LIN {X 0,Y 368.899,Z 889.348,A -85,B 0,C 180,E1 -12566.461,E2 -12566.461} C_VEL
LIN {X 0,Y 368.899,Z 889.344,A -85,B 0,C 180,E1 -12569.043,E2 -12569.043} C_VEL
LIN {X 0,Y 368.91,Z 889.341,A -85,B 0,C 180,E1 -12571.557,E2 -12571.557} C_VEL
LIN {X 0,Y 368.887,Z 889.347,A -85,B 0,C 180,E1 -12575.219,E2 -12575.219} C_VEL
LIN {X 0,Y 368.898,Z 889.343,A -85,B 0,C 180,E1 -12577.602,E2 -12577.602} C_VEL
LIN {X 0,Y 368.909,Z 889.346,A -85,B 0,C 180,E1 -12581.103,E2 -12581.103} C_VEL
LIN {X 0,Y 368.931,Z 889.338,A -85,B 0,C 180,E1 -12584.532,E2 -12584.532} C_VEL
LIN {X 0,Y 369.059,Z 889.323,A -85,B 0,C 180,E1 -12586.79,E2 -12586.79} C_VEL
LIN {X 0,Y 369.059,Z 889.323,A -85,B 0,C 180,E1 -12590.131,E2 -12590.131} C_VEL
LIN {X 0,Y 369.157,Z 889.313,A -85,B 0,C 180,E1 -12593.44,E2 -12593.44} C_VEL
LIN {X 0,Y 369.292,Z 889.298,A -85,B 0,C 180,E1 -12597.818,E2 -12597.818} C_VEL
LIN {X 0,Y 369.204,Z 889.304,A -85,B 0,C 180,E1 -12601.09,E2 -12601.09} C_VEL
LIN {X 0,Y 369.292,Z 889.299,A -85,B 0,C 180,E1 -12602.181,E2 -12602.181} C_VEL
LIN {X 0,Y 369.157,Z 889.314,A -85,B 0,C 180,E1 -12606.559,E2 -12606.559} C_VEL
LIN {X 0,Y 369.058,Z 889.323,A -85,B 0,C 180,E1 -12609.868,E2 -12609.868} C_VEL
LIN {X 0,Y 369.04,Z 889.324,A -85,B 0,C 180,E1 -12613.772,E2 -12613.772} C_VEL
LIN {X 0,Y 368.955,Z 889.335,A -85,B 0,C 180,E1 -12617.744,E2 -12617.744} C_VEL
LIN {X 0,Y 368.91,Z 889.344,A -85,B 0,C 180,E1 -12621.22,E2 -12621.22} C_VEL
LIN {X 0,Y 368.906,Z 889.341,A -85,B 0,C 180,E1 -12623.872,E2 -12623.872} C_VEL
LIN {X 0,Y 368.856,Z 889.354,A -85,B 0,C 180,E1 -12627.212,E2 -12627.212} C_VEL
LIN {X 0,Y 368.892,Z 889.346,A -85,B 0,C 180,E1 -12629.692,E2 -12629.692} C_VEL
LIN {X 0,Y 368.895,Z 889.345,A -85,B 0,C 180,E1 -12633.042,E2 -12633.042} C_VEL
LIN {X 0,Y 368.91,Z 889.342,A -85,B 0,C 180,E1 -12636.197,E2 -12636.197} C_VEL
LIN {X 0,Y 368.872,Z 889.345,A -85,B 0,C 180,E1 -12638.957,E2 -12638.957} C_VEL
LIN {X 0,Y 368.858,Z 889.353,A -85,B 0,C 180,E1 -12642.005,E2 -12642.005} C_VEL
LIN {X 0,Y 368.872,Z 889.345,A -85,B 0,C 180,E1 -12645.174,E2 -12645.174} C_VEL
LIN {X 0,Y 368.86,Z 889.354,A -85,B 0,C 180,E1 -12648.174,E2 -12648.174} C_VEL
LIN {X 0,Y 368.873,Z 889.345,A -85,B 0,C 180,E1 -12651.366,E2 -12651.366} C_VEL
LIN {X 0,Y 368.931,Z 889.339,A -85,B 0,C 180,E1 -12655.145,E2 -12655.145} C_VEL
LIN {X 0,Y 368.895,Z 889.345,A -85,B 0,C 180,E1 -12659.043,E2 -12659.043} C_VEL
LIN {X 0,Y 368.883,Z 889.35,A -85,B 0,C 180,E1 -12662.79,E2 -12662.79} C_VEL
LIN {X 0,Y 368.943,Z 889.489,A -85,B 0,C 180,E1 -12663.316,E2 -12663.316} C_VEL
LIN {X 0,Y 371.115,Z 901.236,A -85,B 0,C 180,E1 -12666.566,E2 -12666.566} C_VEL
LIN {X 0,Y 370.607,Z 910.137,A -85,B 0,C 180,E1 -12668.881,E2 -12668.881} C_VEL
LIN {X 0,Y 369.569,Z 923.419,A -85,B 0,C 180,E1 -12672.286,E2 -12672.286} C_VEL
LIN {X 0,Y 369.237,Z 928.5,A -85,B 0,C 180,E1 -12673.547,E2 -12673.547} C_VEL
LIN {X 0,Y 372.227,Z 955.937,A -85,B 0,C 180,E1 -12674.334,E2 -12674.334} C_VEL
LIN {X 0,Y 371.384,Z 1006.743,A -85,B 0,C 180,E1 -12675.583,E2 -12675.583} C_VEL
LIN {X 0,Y 370.796,Z 1018.982,A -85,B 0,C 180,E1 -12676.085,E2 -12676.085} C_VEL
LIN {X 0,Y 370.446,Z 1028.911,A -85,B 0,C 180,E1 -12676.701,E2 -12676.701} C_VEL
LIN {X 0,Y 369.98,Z 1037.486,A -85,B 0,C 180,E1 -12677.382,E2 -12677.382} C_VEL
LIN {X 0,Y 369.472,Z 1045.773,A -85,B 0,C 180,E1 -12678.2,E2 -12678.2} C_VEL
LIN {X 0,Y 369.082,Z 1052.645,A -85,B 0,C 180,E1 -12679.023,E2 -12679.023} C_VEL
LIN {X 0,Y 368.68,Z 1058.484,A -85,B 0,C 180,E1 -12679.844,E2 -12679.844} C_VEL
LIN {X 0,Y 368.286,Z 1065.014,A -85,B 0,C 180,E1 -12680.942,E2 -12680.942} C_VEL
LIN {X 0,Y 367.983,Z 1070.432,A -85,B 0,C 180,E1 -12682.041,E2 -12682.041} C_VEL
LIN {X 0,Y 367.732,Z 1075.925,A -85,B 0,C 180,E1 -12683.415,E2 -12683.415} C_VEL
LIN {X 0,Y 367.595,Z 1081.012,A -85,B 0,C 180,E1 -12685.064,E2 -12685.064} C_VEL
LIN {X 0,Y 367.435,Z 1084.496,A -85,B 0,C 180,E1 -12686.71,E2 -12686.71} C_VEL
LIN {X 0,Y 367.453,Z 1086.131,A -85,B 0,C 180,E1 -12687.808,E2 -12687.808} C_VEL
LIN {X 0,Y 367.538,Z 1087.133,A -85,B 0,C 180,E1 -12688.904,E2 -12688.904} C_VEL
LIN {X 0,Y 367.52,Z 1087.577,A -85,B 0,C 180,E1 -12690,E2 -12690} C_VEL
LIN {X 0,Y 367.484,Z 1087.506,A -85,B 0,C 180,E1 -12691.096,E2 -12691.096} C_VEL
LIN {X 0,Y 367.412,Z 1086.92,A -85,B 0,C 180,E1 -12692.192,E2 -12692.192} C_VEL
LIN {X 0,Y 367.428,Z 1085.796,A -85,B 0,C 180,E1 -12693.289,E2 -12693.289} C_VEL
LIN {X 0,Y 367.571,Z 1082.946,A -85,B 0,C 180,E1 -12694.936,E2 -12694.936} C_VEL
LIN {X 0,Y 367.685,Z 1079.551,A -85,B 0,C 180,E1 -12696.315,E2 -12696.315} C_VEL
LIN {X 0,Y 367.978,Z 1075.132,A -85,B 0,C 180,E1 -12697.683,E2 -12697.683} C_VEL
LIN {X 0,Y 368.342,Z 1069.514,A -85,B 0,C 180,E1 -12699.056,E2 -12699.056} C_VEL
LIN {X 0,Y 368.948,Z 1062.566,A -85,B 0,C 180,E1 -12700.426,E2 -12700.426} C_VEL
LIN {X 0,Y 369.746,Z 1053.734,A -85,B 0,C 180,E1 -12701.79,E2 -12701.79} C_VEL
LIN {X 0,Y 370.374,Z 1046.059,A -85,B 0,C 180,E1 -12702.743,E2 -12702.743} C_VEL
LIN {X 0,Y 370.978,Z 1038.109,A -85,B 0,C 180,E1 -12703.558,E2 -12703.558} C_VEL
LIN {X 0,Y 371.559,Z 1030.04,A -85,B 0,C 180,E1 -12704.235,E2 -12704.235} C_VEL
LIN {X 0,Y 372.224,Z 1020.928,A -85,B 0,C 180,E1 -12704.837,E2 -12704.837} C_VEL
LIN {X 0,Y 372.916,Z 1010.324,A -85,B 0,C 180,E1 -12705.359,E2 -12705.359} C_VEL
LIN {X 0,Y 373.461,Z 995.486,A -85,B 0,C 180,E1 -12705.821,E2 -12705.821} C_VEL
LIN {X 0,Y 374.43,Z 954.567,A -85,B 0,C 180,E1 -12706.913,E2 -12706.913} C_VEL
LIN {X 0,Y 372.829,Z 940.302,A -85,B 0,C 180,E1 -12707.443,E2 -12707.443} C_VEL
LIN {X 0,Y 370.066,Z 925.912,A -85,B 0,C 180,E1 -12708.097,E2 -12708.097} C_VEL
LIN {X 0,Y 371.647,Z 911.366,A -85,B 0,C 180,E1 -12712.088,E2 -12712.088} C_VEL
LIN {X 0,Y 372.127,Z 906.885,A -85,B 0,C 180,E1 -12713.366,E2 -12713.366} C_VEL
LIN {X 0,Y 371.437,Z 901.089,A -85,B 0,C 180,E1 -12715.211,E2 -12715.211} C_VEL
LIN {X 0,Y 369.934,Z 893.844,A -85,B 0,C 180,E1 -12717.739,E2 -12717.739} C_VEL
LIN {X 0,Y 368.863,Z 889.353,A -85,B 0,C 180,E1 -12719.507,E2 -12719.507} C_VEL
LIN {X 0,Y 368.894,Z 889.349,A -85,B 0,C 180,E1 -12722.238,E2 -12722.238} C_VEL
LIN {X 0,Y 368.92,Z 889.346,A -85,B 0,C 180,E1 -12725,E2 -12725} C_VEL
LIN {X 0,Y 368.871,Z 889.35,A -85,B 0,C 180,E1 -12728.634,E2 -12728.634} C_VEL
LIN {X 0,Y 368.855,Z 889.351,A -85,B 0,C 180,E1 -12732.005,E2 -12732.005} C_VEL
LIN {X 0,Y 368.87,Z 889.349,A -85,B 0,C 180,E1 -12735.175,E2 -12735.175} C_VEL
LIN {X 0,Y 368.858,Z 889.352,A -85,B 0,C 180,E1 -12738.175,E2 -12738.175} C_VEL
LIN {X 0,Y 368.872,Z 889.349,A -85,B 0,C 180,E1 -12741.367,E2 -12741.367} C_VEL
LIN {X 0,Y 368.928,Z 889.341,A -85,B 0,C 180,E1 -12745.146,E2 -12745.146} C_VEL
LIN {X 0,Y 368.894,Z 889.347,A -85,B 0,C 180,E1 -12749.044,E2 -12749.044} C_VEL
LIN {X 0,Y 368.904,Z 889.345,A -85,B 0,C 180,E1 -12751.558,E2 -12751.558} C_VEL
LIN {X 0,Y 368.882,Z 889.354,A -85,B 0,C 180,E1 -12755.22,E2 -12755.22} C_VEL
LIN {X 0,Y 368.946,Z 889.49,A -85,B 0,C 180,E1 -12756.569,E2 -12756.569} C_VEL
LIN {X 0,Y 370.273,Z 896.019,A -85,B 0,C 180,E1 -12759.443,E2 -12759.443} C_VEL
LIN {X 0,Y 370.863,Z 900.746,A -85,B 0,C 180,E1 -12761.356,E2 -12761.356} C_VEL
LIN {X 0,Y 370.818,Z 902.644,A -85,B 0,C 180,E1 -12762.048,E2 -12762.048} C_VEL
LIN {X 0,Y 374.529,Z 916.761,A -85,B 0,C 180,E1 -12762.768,E2 -12762.768} C_VEL
LIN {X 0,Y 375.198,Z 921.412,A -85,B 0,C 180,E1 -12762.953,E2 -12762.953} C_VEL
LIN {X 0,Y 373.379,Z 979.291,A -85,B 0,C 180,E1 -12764.527,E2 -12764.527} C_VEL
LIN {X 0,Y 372.923,Z 991.072,A -85,B 0,C 180,E1 -12765.052,E2 -12765.052} C_VEL
LIN {X 0,Y 372.29,Z 1000.633,A -85,B 0,C 180,E1 -12765.655,E2 -12765.655} C_VEL
LIN {X 0,Y 371.8,Z 1008.981,A -85,B 0,C 180,E1 -12766.333,E2 -12766.333} C_VEL
LIN {X 0,Y 371.247,Z 1017.092,A -85,B 0,C 180,E1 -12767.148,E2 -12767.148} C_VEL
LIN {X 0,Y 370.556,Z 1024.861,A -85,B 0,C 180,E1 -12768.097,E2 -12768.097} C_VEL
LIN {X 0,Y 370.044,Z 1031.287,A -85,B 0,C 180,E1 -12769.052,E2 -12769.052} C_VEL
LIN {X 0,Y 369.282,Z 1038.862,A -85,B 0,C 180,E1 -12770.415,E2 -12770.415} C_VEL
LIN {X 0,Y 368.76,Z 1044.799,A -85,B 0,C 180,E1 -12771.783,E2 -12771.783} C_VEL
LIN {X 0,Y 368.34,Z 1050.206,A -85,B 0,C 180,E1 -12773.427,E2 -12773.427} C_VEL
LIN {X 0,Y 367.932,Z 1053.048,A -85,B 0,C 180,E1 -12774.52,E2 -12774.52} C_VEL
LIN {X 0,Y 367.798,Z 1055.276,A -85,B 0,C 180,E1 -12775.617,E2 -12775.617} C_VEL
LIN {X 0,Y 367.766,Z 1056.891,A -85,B 0,C 180,E1 -12776.714,E2 -12776.714} C_VEL
LIN {X 0,Y 367.665,Z 1057.898,A -85,B 0,C 180,E1 -12777.81,E2 -12777.81} C_VEL
LIN {X 0,Y 367.551,Z 1058.387,A -85,B 0,C 180,E1 -12778.905,E2 -12778.905} C_VEL
LIN {X 0,Y 367.504,Z 1058.367,A -85,B 0,C 180,E1 -12780.001,E2 -12780.001} C_VEL
LIN {X 0,Y 367.497,Z 1057.838,A -85,B 0,C 180,E1 -12781.096,E2 -12781.096} C_VEL
LIN {X 0,Y 367.517,Z 1056.751,A -85,B 0,C 180,E1 -12782.192,E2 -12782.192} C_VEL
LIN {X 0,Y 367.588,Z 1053.997,A -85,B 0,C 180,E1 -12783.837,E2 -12783.837} C_VEL
LIN {X 0,Y 367.744,Z 1051.48,A -85,B 0,C 180,E1 -12784.934,E2 -12784.934} C_VEL
LIN {X 0,Y 367.989,Z 1046.335,A -85,B 0,C 180,E1 -12786.581,E2 -12786.581} C_VEL
LIN {X 0,Y 368.218,Z 1042.025,A -85,B 0,C 180,E1 -12787.679,E2 -12787.679} C_VEL
LIN {X 0,Y 368.466,Z 1036.826,A -85,B 0,C 180,E1 -12788.778,E2 -12788.778} C_VEL
LIN {X 0,Y 368.906,Z 1030.558,A -85,B 0,C 180,E1 -12789.873,E2 -12789.873} C_VEL
LIN {X 0,Y 369.373,Z 1022.942,A -85,B 0,C 180,E1 -12790.969,E2 -12790.969} C_VEL
LIN {X 0,Y 369.855,Z 1014.814,A -85,B 0,C 180,E1 -12791.926,E2 -12791.926} C_VEL
LIN {X 0,Y 370.421,Z 1004.687,A -85,B 0,C 180,E1 -12792.882,E2 -12792.882} C_VEL
LIN {X 0,Y 370.87,Z 993.951,A -85,B 0,C 180,E1 -12793.633,E2 -12793.633} C_VEL
LIN {X 0,Y 371.104,Z 984.065,A -85,B 0,C 180,E1 -12794.148,E2 -12794.148} C_VEL
LIN {X 0,Y 371.472,Z 973.564,A -85,B 0,C 180,E1 -12794.518,E2 -12794.518} C_VEL
LIN {X 0,Y 372.416,Z 918.799,A -85,B 0,C 180,E1 -12795.838,E2 -12795.838} C_VEL
LIN {X 0,Y 369.303,Z 899.54,A -85,B 0,C 180,E1 -12796.448,E2 -12796.448} C_VEL
LIN {X 0,Y 369.477,Z 893.53,A -85,B 0,C 180,E1 -12798.363,E2 -12798.363} C_VEL
LIN {X 0,Y 369.004,Z 889.33,A -85,B 0,C 180,E1 -12799.76,E2 -12799.76} C_VEL
LIN {X 0,Y 368.906,Z 889.341,A -85,B 0,C 180,E1 -12803.873,E2 -12803.873} C_VEL
LIN {X 0,Y 368.857,Z 889.354,A -85,B 0,C 180,E1 -12807.213,E2 -12807.213} C_VEL
LIN {X 0,Y 368.893,Z 889.346,A -85,B 0,C 180,E1 -12809.693,E2 -12809.693} C_VEL
LIN {X 0,Y 368.897,Z 889.344,A -85,B 0,C 180,E1 -12813.043,E2 -12813.043} C_VEL
LIN {X 0,Y 368.913,Z 889.341,A -85,B 0,C 180,E1 -12816.198,E2 -12816.198} C_VEL
LIN {X 0,Y 368.874,Z 889.345,A -85,B 0,C 180,E1 -12818.958,E2 -12818.958} C_VEL
LIN {X 0,Y 368.86,Z 889.352,A -85,B 0,C 180,E1 -12822.006,E2 -12822.006} C_VEL
LIN {X 0,Y 368.874,Z 889.345,A -85,B 0,C 180,E1 -12825.175,E2 -12825.175} C_VEL
LIN {X 0,Y 368.863,Z 889.353,A -85,B 0,C 180,E1 -12828.175,E2 -12828.175} C_VEL
LIN {X 0,Y 368.877,Z 889.345,A -85,B 0,C 180,E1 -12831.367,E2 -12831.367} C_VEL
LIN {X 0,Y 368.934,Z 889.338,A -85,B 0,C 180,E1 -12835.146,E2 -12835.146} C_VEL
LIN {X 0,Y 368.899,Z 889.344,A -85,B 0,C 180,E1 -12839.044,E2 -12839.044} C_VEL
LIN {X 0,Y 368.91,Z 889.341,A -85,B 0,C 180,E1 -12841.558,E2 -12841.558} C_VEL
LIN {X 0,Y 368.925,Z 889.342,A -85,B 0,C 180,E1 -12845.222,E2 -12845.222} C_VEL
LIN {X 0,Y 368.924,Z 889.344,A -85,B 0,C 180,E1 -12848.981,E2 -12848.981} C_VEL
LIN {X 0,Y 368.957,Z 889.335,A -85,B 0,C 180,E1 -12852.256,E2 -12852.256} C_VEL
LIN {X 0,Y 369.017,Z 889.331,A -85,B 0,C 180,E1 -12855.665,E2 -12855.665} C_VEL
LIN {X 0,Y 369.013,Z 889.33,A -85,B 0,C 180,E1 -12859.021,E2 -12859.021} C_VEL
LIN {X 0,Y 369.12,Z 889.315,A -85,B 0,C 180,E1 -12862.341,E2 -12862.341} C_VEL
LIN {X 0,Y 369.117,Z 889.315,A -85,B 0,C 180,E1 -12864.537,E2 -12864.537} C_VEL
LIN {X 0,Y 369.295,Z 889.298,A -85,B 0,C 180,E1 -12867.819,E2 -12867.819} C_VEL
LIN {X 0,Y 369.206,Z 889.304,A -85,B 0,C 180,E1 -12871.091,E2 -12871.091} C_VEL
LIN {X 0,Y 369.294,Z 889.299,A -85,B 0,C 180,E1 -12872.182,E2 -12872.182} C_VEL
LIN {X 0,Y 369.159,Z 889.314,A -85,B 0,C 180,E1 -12876.559,E2 -12876.559} C_VEL
LIN {X 0,Y 369.061,Z 889.323,A -85,B 0,C 180,E1 -12879.869,E2 -12879.869} C_VEL
LIN {X 0,Y 369.043,Z 889.324,A -85,B 0,C 180,E1 -12883.772,E2 -12883.772} C_VEL
LIN {X 0,Y 368.958,Z 889.334,A -85,B 0,C 180,E1 -12887.745,E2 -12887.745} C_VEL
LIN {X 0,Y 368.913,Z 889.344,A -85,B 0,C 180,E1 -12891.221,E2 -12891.221} C_VEL
LIN {X 0,Y 368.909,Z 889.341,A -85,B 0,C 180,E1 -12893.872,E2 -12893.872} C_VEL
LIN {X 0,Y 368.86,Z 889.353,A -85,B 0,C 180,E1 -12897.212,E2 -12897.212} C_VEL
LIN {X 0,Y 368.896,Z 889.345,A -85,B 0,C 180,E1 -12899.692,E2 -12899.692} C_VEL
LIN {X 0,Y 368.9,Z 889.344,A -85,B 0,C 180,E1 -12903.042,E2 -12903.042} C_VEL
LIN {X 0,Y 368.89,Z 889.344,A -85,B 0,C 180,E1 -12904.117,E2 -12904.117} C_VEL
LIN {X 0,Y 368.239,Z 889.427,A -85,B 0,C 180,E1 -12905.029,E2 -12905.029} C_VEL
LIN {X 0,Y 365.381,Z 889.78,A -85,B 0,C 180,E1 -12906.512,E2 -12906.512} C_VEL
LIN {X 0,Y 362.952,Z 890.09,A -85,B 0,C 180,E1 -12907.711,E2 -12907.711} C_VEL
LIN {X 0,Y 361.911,Z 890.213,A -85,B 0,C 180,E1 -12908.639,E2 -12908.639} C_VEL
LIN {X 0,Y 361.829,Z 890.223,A -85,B 0,C 180,E1 -12908.953,E2 -12908.953} C_VEL
LIN {X 0,Y 361.833,Z 890.222,A -85,B 0,C 180,E1 -12912.83,E2 -12912.83} C_VEL
LIN {X 0,Y 361.817,Z 890.229,A -85,B 0,C 180,E1 -12915.947,E2 -12915.947} C_VEL
LIN {X 0,Y 361.813,Z 890.224,A -85,B 0,C 180,E1 -12919.249,E2 -12919.249} C_VEL
LIN {X 0,Y 361.864,Z 890.219,A -85,B 0,C 180,E1 -12922.981,E2 -12922.981} C_VEL
LIN {X 0,Y 361.861,Z 890.224,A -85,B 0,C 180,E1 -12926.631,E2 -12926.631} C_VEL
LIN {X 0,Y 361.85,Z 890.22,A -85,B 0,C 180,E1 -12929.669,E2 -12929.669} C_VEL
LIN {X 0,Y 361.857,Z 890.22,A -85,B 0,C 180,E1 -12933.467,E2 -12933.467} C_VEL
LIN {X 0,Y 361.863,Z 890.224,A -85,B 0,C 180,E1 -12937.142,E2 -12937.142} C_VEL
LIN {X 0,Y 361.849,Z 890.222,A -85,B 0,C 180,E1 -12940.72,E2 -12940.72} C_VEL
LIN {X 0,Y 361.89,Z 890.219,A -85,B 0,C 180,E1 -12943.063,E2 -12943.063} C_VEL
LIN {X 0,Y 362.002,Z 890.201,A -85,B 0,C 180,E1 -12946.527,E2 -12946.527} C_VEL
LIN {X 0,Y 361.996,Z 890.205,A -85,B 0,C 180,E1 -12949.936,E2 -12949.936} C_VEL
LIN {X 0,Y 362.121,Z 890.189,A -85,B 0,C 180,E1 -12953.312,E2 -12953.312} C_VEL
LIN {X 0,Y 362.254,Z 890.175,A -85,B 0,C 180,E1 -12957.776,E2 -12957.776} C_VEL
LIN {X 0,Y 362.175,Z 890.179,A -85,B 0,C 180,E1 -12961.111,E2 -12961.111} C_VEL
LIN {X 0,Y 362.254,Z 890.175,A -85,B 0,C 180,E1 -12962.223,E2 -12962.223} C_VEL
LIN {X 0,Y 362.121,Z 890.189,A -85,B 0,C 180,E1 -12966.687,E2 -12966.687} C_VEL
LIN {X 0,Y 361.995,Z 890.205,A -85,B 0,C 180,E1 -12970.063,E2 -12970.063} C_VEL
LIN {X 0,Y 361.982,Z 890.204,A -85,B 0,C 180,E1 -12973.886,E2 -12973.886} C_VEL
LIN {X 0,Y 361.886,Z 890.216,A -85,B 0,C 180,E1 -12978.103,E2 -12978.103} C_VEL
LIN {X 0,Y 361.853,Z 890.22,A -85,B 0,C 180,E1 -12981.655,E2 -12981.655} C_VEL
LIN {X 0,Y 361.859,Z 890.224,A -85,B 0,C 180,E1 -12985.295,E2 -12985.295} C_VEL
LIN {X 0,Y 361.856,Z 890.223,A -85,B 0,C 180,E1 -12989.073,E2 -12989.073} C_VEL
LIN {X 0,Y 361.847,Z 890.222,A -85,B 0,C 180,E1 -12992.944,E2 -12992.944} C_VEL
LIN {X 0,Y 361.863,Z 890.225,A -85,B 0,C 180,E1 -12995.637,E2 -12995.637} C_VEL
LIN {X 0,Y 361.824,Z 890.224,A -85,B 0,C 180,E1 -12999.017,E2 -12999.017} C_VEL
LIN {X 0,Y 361.828,Z 890.223,A -85,B 0,C 180,E1 -13002.83,E2 -13002.83} C_VEL
LIN {X 0,Y 361.813,Z 890.23,A -85,B 0,C 180,E1 -13005.947,E2 -13005.947} C_VEL
LIN {X 0,Y 361.809,Z 890.225,A -85,B 0,C 180,E1 -13009.249,E2 -13009.249} C_VEL
LIN {X 0,Y 361.86,Z 890.22,A -85,B 0,C 180,E1 -13012.981,E2 -13012.981} C_VEL
LIN {X 0,Y 361.856,Z 890.225,A -85,B 0,C 180,E1 -13016.631,E2 -13016.631} C_VEL
LIN {X 0,Y 361.845,Z 890.22,A -85,B 0,C 180,E1 -13019.669,E2 -13019.669} C_VEL
LIN {X 0,Y 361.879,Z 890.287,A -85,B 0,C 180,E1 -13023.145,E2 -13023.145} C_VEL
LIN {X 0,Y 364.001,Z 901.747,A -85,B 0,C 180,E1 -13026.382,E2 -13026.382} C_VEL
LIN {X 0,Y 363.896,Z 906.742,A -85,B 0,C 180,E1 -13027.718,E2 -13027.718} C_VEL
LIN {X 0,Y 362.776,Z 920.524,A -85,B 0,C 180,E1 -13031.332,E2 -13031.332} C_VEL
LIN {X 0,Y 362.246,Z 928.09,A -85,B 0,C 180,E1 -13033.3,E2 -13033.3} C_VEL
LIN {X 0,Y 365.281,Z 955.565,A -85,B 0,C 180,E1 -13034.116,E2 -13034.116} C_VEL
LIN {X 0,Y 364.371,Z 1006.424,A -85,B 0,C 180,E1 -13035.413,E2 -13035.413} C_VEL
LIN {X 0,Y 363.82,Z 1017.855,A -85,B 0,C 180,E1 -13035.884,E2 -13035.884} C_VEL
LIN {X 0,Y 363.4,Z 1028.918,A -85,B 0,C 180,E1 -13036.58,E2 -13036.58} C_VEL
LIN {X 0,Y 362.924,Z 1037.423,A -85,B 0,C 180,E1 -13037.274,E2 -13037.274} C_VEL
LIN {X 0,Y 362.418,Z 1045.665,A -85,B 0,C 180,E1 -13038.109,E2 -13038.109} C_VEL
LIN {X 0,Y 362.017,Z 1052.505,A -85,B 0,C 180,E1 -13038.947,E2 -13038.947} C_VEL
LIN {X 0,Y 361.548,Z 1059.189,A -85,B 0,C 180,E1 -13039.924,E2 -13039.924} C_VEL
LIN {X 0,Y 361.158,Z 1065.557,A -85,B 0,C 180,E1 -13041.044,E2 -13041.044} C_VEL
LIN {X 0,Y 360.886,Z 1070.836,A -85,B 0,C 180,E1 -13042.165,E2 -13042.165} C_VEL
LIN {X 0,Y 360.693,Z 1075.211,A -85,B 0,C 180,E1 -13043.286,E2 -13043.286} C_VEL
LIN {X 0,Y 360.51,Z 1080.389,A -85,B 0,C 180,E1 -13044.967,E2 -13044.967} C_VEL
LIN {X 0,Y 360.356,Z 1084.025,A -85,B 0,C 180,E1 -13046.646,E2 -13046.646} C_VEL
LIN {X 0,Y 360.359,Z 1085.689,A -85,B 0,C 180,E1 -13047.764,E2 -13047.764} C_VEL
LIN {X 0,Y 360.454,Z 1086.735,A -85,B 0,C 180,E1 -13048.883,E2 -13048.883} C_VEL
LIN {X 0,Y 360.456,Z 1087.245,A -85,B 0,C 180,E1 -13050,E2 -13050} C_VEL
LIN {X 0,Y 360.385,Z 1087.233,A -85,B 0,C 180,E1 -13051.117,E2 -13051.117} C_VEL
LIN {X 0,Y 360.314,Z 1086.702,A -85,B 0,C 180,E1 -13052.235,E2 -13052.235} C_VEL
LIN {X 0,Y 360.348,Z 1085.596,A -85,B 0,C 180,E1 -13053.354,E2 -13053.354} C_VEL
LIN {X 0,Y 360.488,Z 1082.825,A -85,B 0,C 180,E1 -13055.033,E2 -13055.033} C_VEL
LIN {X 0,Y 360.666,Z 1078.695,A -85,B 0,C 180,E1 -13056.714,E2 -13056.714} C_VEL
LIN {X 0,Y 360.999,Z 1074.143,A -85,B 0,C 180,E1 -13058.114,E2 -13058.114} C_VEL
LIN {X 0,Y 361.479,Z 1068.4,A -85,B 0,C 180,E1 -13059.512,E2 -13059.512} C_VEL
LIN {X 0,Y 362.14,Z 1061.248,A -85,B 0,C 180,E1 -13060.907,E2 -13060.907} C_VEL
LIN {X 0,Y 362.947,Z 1052.036,A -85,B 0,C 180,E1 -13062.298,E2 -13062.298} C_VEL
LIN {X 0,Y 363.677,Z 1044.075,A -85,B 0,C 180,E1 -13063.266,E2 -13063.266} C_VEL
LIN {X 0,Y 364.446,Z 1034.341,A -85,B 0,C 180,E1 -13064.233,E2 -13064.233} C_VEL
LIN {X 0,Y 365.322,Z 1023.496,A -85,B 0,C 180,E1 -13065.053,E2 -13065.053} C_VEL
LIN {X 0,Y 366.111,Z 1013.024,A -85,B 0,C 180,E1 -13065.623,E2 -13065.623} C_VEL
LIN {X 0,Y 366.578,Z 1003.239,A -85,B 0,C 180,E1 -13066.007,E2 -13066.007} C_VEL
LIN {X 0,Y 367.916,Z 955.498,A -85,B 0,C 180,E1 -13067.329,E2 -13067.329} C_VEL
LIN {X 0,Y 366.449,Z 941.662,A -85,B 0,C 180,E1 -13067.87,E2 -13067.87} C_VEL
LIN {X 0,Y 363.843,Z 928.167,A -85,B 0,C 180,E1 -13068.508,E2 -13068.508} C_VEL
LIN {X 0,Y 363.285,Z 925.477,A -85,B 0,C 180,E1 -13068.664,E2 -13068.664} C_VEL
LIN {X 0,Y 364.942,Z 911.374,A -85,B 0,C 180,E1 -13072.653,E2 -13072.653} C_VEL
LIN {X 0,Y 365.222,Z 907.458,A -85,B 0,C 180,E1 -13073.835,E2 -13073.835} C_VEL
LIN {X 0,Y 364.427,Z 901.823,A -85,B 0,C 180,E1 -13075.715,E2 -13075.715} C_VEL
LIN {X 0,Y 362.904,Z 894.732,A -85,B 0,C 180,E1 -13078.324,E2 -13078.324} C_VEL
LIN {X 0,Y 361.839,Z 890.227,A -85,B 0,C 180,E1 -13080.17,E2 -13080.17} C_VEL
LIN {X 0,Y 361.855,Z 890.227,A -85,B 0,C 180,E1 -13083.369,E2 -13083.369} C_VEL
LIN {X 0,Y 361.857,Z 890.224,A -85,B 0,C 180,E1 -13087.019,E2 -13087.019} C_VEL
LIN {X 0,Y 361.807,Z 890.227,A -85,B 0,C 180,E1 -13090.751,E2 -13090.751} C_VEL
LIN {X 0,Y 361.809,Z 890.231,A -85,B 0,C 180,E1 -13094.37,E2 -13094.37} C_VEL
LIN {X 0,Y 361.82,Z 890.227,A -85,B 0,C 180,E1 -13097.571,E2 -13097.571} C_VEL
LIN {X 0,Y 361.838,Z 890.226,A -85,B 0,C 180,E1 -13101.572,E2 -13101.572} C_VEL
LIN {X 0,Y 361.868,Z 890.222,A -85,B 0,C 180,E1 -13104.657,E2 -13104.657} C_VEL
LIN {X 0,Y 361.835,Z 890.227,A -85,B 0,C 180,E1 -13108.371,E2 -13108.371} C_VEL
LIN {X 0,Y 361.847,Z 890.226,A -85,B 0,C 180,E1 -13110.951,E2 -13110.951} C_VEL
LIN {X 0,Y 361.857,Z 890.227,A -85,B 0,C 180,E1 -13114.705,E2 -13114.705} C_VEL
LIN {X 0,Y 361.886,Z 890.418,A -85,B 0,C 180,E1 -13115.932,E2 -13115.932} C_VEL
LIN {X 0,Y 363.302,Z 897.119,A -85,B 0,C 180,E1 -13119.031,E2 -13119.031} C_VEL
LIN {X 0,Y 363.99,Z 902.06,A -85,B 0,C 180,E1 -13121.103,E2 -13121.103} C_VEL
LIN {X 0,Y 363.981,Z 903.044,A -85,B 0,C 180,E1 -13121.488,E2 -13121.488} C_VEL
LIN {X 0,Y 367.562,Z 915.604,A -85,B 0,C 180,E1 -13122.198,E2 -13122.198} C_VEL
LIN {X 0,Y 368.772,Z 921.813,A -85,B 0,C 180,E1 -13122.492,E2 -13122.492} C_VEL
LIN {X 0,Y 366.755,Z 980.697,A -85,B 0,C 180,E1 -13124.154,E2 -13124.154} C_VEL
LIN {X 0,Y 366.287,Z 992.208,A -85,B 0,C 180,E1 -13124.703,E2 -13124.703} C_VEL
LIN {X 0,Y 365.566,Z 1002.438,A -85,B 0,C 180,E1 -13125.385,E2 -13125.385} C_VEL
LIN {X 0,Y 364.916,Z 1011.91,A -85,B 0,C 180,E1 -13126.212,E2 -13126.212} C_VEL
LIN {X 0,Y 364.076,Z 1021.861,A -85,B 0,C 180,E1 -13127.316,E2 -13127.316} C_VEL
LIN {X 0,Y 363.31,Z 1030.516,A -85,B 0,C 180,E1 -13128.564,E2 -13128.564} C_VEL
LIN {X 0,Y 362.618,Z 1036.852,A -85,B 0,C 180,E1 -13129.673,E2 -13129.673} C_VEL
LIN {X 0,Y 362.121,Z 1042.099,A -85,B 0,C 180,E1 -13130.787,E2 -13130.787} C_VEL
LIN {X 0,Y 361.786,Z 1045.497,A -85,B 0,C 180,E1 -13131.623,E2 -13131.623} C_VEL
LIN {X 0,Y 361.42,Z 1049.962,A -85,B 0,C 180,E1 -13132.982,E2 -13132.982} C_VEL
LIN {X 0,Y 360.899,Z 1053.596,A -85,B 0,C 180,E1 -13134.413,E2 -13134.413} C_VEL
LIN {X 0,Y 360.73,Z 1055.75,A -85,B 0,C 180,E1 -13135.531,E2 -13135.531} C_VEL
LIN {X 0,Y 360.699,Z 1057.33,A -85,B 0,C 180,E1 -13136.649,E2 -13136.649} C_VEL
LIN {X 0,Y 360.591,Z 1058.296,A -85,B 0,C 180,E1 -13137.767,E2 -13137.767} C_VEL
LIN {X 0,Y 360.472,Z 1058.722,A -85,B 0,C 180,E1 -13138.883,E2 -13138.883} C_VEL
LIN {X 0,Y 360.423,Z 1058.638,A -85,B 0,C 180,E1 -13140.001,E2 -13140.001} C_VEL
LIN {X 0,Y 360.4,Z 1058.044,A -85,B 0,C 180,E1 -13141.118,E2 -13141.118} C_VEL
LIN {X 0,Y 360.42,Z 1056.916,A -85,B 0,C 180,E1 -13142.236,E2 -13142.236} C_VEL
LIN {X 0,Y 360.514,Z 1054.049,A -85,B 0,C 180,E1 -13143.913,E2 -13143.913} C_VEL
LIN {X 0,Y 360.715,Z 1049.844,A -85,B 0,C 180,E1 -13145.591,E2 -13145.591} C_VEL
LIN {X 0,Y 361.049,Z 1044.378,A -85,B 0,C 180,E1 -13147.213,E2 -13147.213} C_VEL
LIN {X 0,Y 361.337,Z 1037.934,A -85,B 0,C 180,E1 -13148.67,E2 -13148.67} C_VEL
LIN {X 0,Y 361.773,Z 1031.811,A -85,B 0,C 180,E1 -13149.787,E2 -13149.787} C_VEL
LIN {X 0,Y 362.24,Z 1024.366,A -85,B 0,C 180,E1 -13150.905,E2 -13150.905} C_VEL
LIN {X 0,Y 362.732,Z 1016.449,A -85,B 0,C 180,E1 -13151.88,E2 -13151.88} C_VEL
LIN {X 0,Y 363.163,Z 1008.15,A -85,B 0,C 180,E1 -13152.717,E2 -13152.717} C_VEL
LIN {X 0,Y 363.666,Z 997.731,A -85,B 0,C 180,E1 -13153.552,E2 -13153.552} C_VEL
LIN {X 0,Y 364.041,Z 986.186,A -85,B 0,C 180,E1 -13154.214,E2 -13154.214} C_VEL
LIN {X 0,Y 364.4,Z 975.683,A -85,B 0,C 180,E1 -13154.622,E2 -13154.622} C_VEL
LIN {X 0,Y 365.486,Z 919.722,A -85,B 0,C 180,E1 -13156.033,E2 -13156.033} C_VEL
LIN {X 0,Y 362.287,Z 899.844,A -85,B 0,C 180,E1 -13156.663,E2 -13156.663} C_VEL
LIN {X 0,Y 362.414,Z 893.862,A -85,B 0,C 180,E1 -13158.603,E2 -13158.603} C_VEL
LIN {X 0,Y 361.979,Z 890.205,A -85,B 0,C 180,E1 -13159.864,E2 -13159.864} C_VEL
LIN {X 0,Y 361.862,Z 890.218,A -85,B 0,C 180,E1 -13164.102,E2 -13164.102} C_VEL
LIN {X 0,Y 361.835,Z 890.223,A -85,B 0,C 180,E1 -13167.786,E2 -13167.786} C_VEL
LIN {X 0,Y 361.849,Z 890.225,A -85,B 0,C 180,E1 -13171.286,E2 -13171.286} C_VEL
LIN {X 0,Y 361.853,Z 890.22,A -85,B 0,C 180,E1 -13174.281,E2 -13174.281} C_VEL
LIN {X 0,Y 361.859,Z 890.221,A -85,B 0,C 180,E1 -13177.222,E2 -13177.222} C_VEL
LIN {X 0,Y 361.812,Z 890.225,A -85,B 0,C 180,E1 -13180.751,E2 -13180.751} C_VEL
LIN {X 0,Y 361.813,Z 890.227,A -85,B 0,C 180,E1 -13184.37,E2 -13184.37} C_VEL
LIN {X 0,Y 361.825,Z 890.225,A -85,B 0,C 180,E1 -13187.571,E2 -13187.571} C_VEL
LIN {X 0,Y 361.843,Z 890.221,A -85,B 0,C 180,E1 -13191.572,E2 -13191.572} C_VEL
LIN {X 0,Y 361.873,Z 890.221,A -85,B 0,C 180,E1 -13194.657,E2 -13194.657} C_VEL
LIN {X 0,Y 361.84,Z 890.225,A -85,B 0,C 180,E1 -13198.371,E2 -13198.371} C_VEL
LIN {X 0,Y 361.869,Z 890.222,A -85,B 0,C 180,E1 -13200.953,E2 -13200.953} C_VEL
LIN {X 0,Y 361.882,Z 890.22,A -85,B 0,C 180,E1 -13204.707,E2 -13204.707} C_VEL
LIN {X 0,Y 361.857,Z 890.22,A -85,B 0,C 180,E1 -13208.345,E2 -13208.345} C_VEL
LIN {X 0,Y 361.908,Z 890.213,A -85,B 0,C 180,E1 -13212.093,E2 -13212.093} C_VEL
LIN {X 0,Y 361.963,Z 890.213,A -85,B 0,C 180,E1 -13215.38,E2 -13215.38} C_VEL
LIN {X 0,Y 361.965,Z 890.206,A -85,B 0,C 180,E1 -13218.804,E2 -13218.804} C_VEL
LIN {X 0,Y 362.082,Z 890.193,A -85,B 0,C 180,E1 -13222.191,E2 -13222.191} C_VEL
LIN {X 0,Y 362.091,Z 890.191,A -85,B 0,C 180,E1 -13224.431,E2 -13224.431} C_VEL
LIN {X 0,Y 362.257,Z 890.174,A -85,B 0,C 180,E1 -13227.776,E2 -13227.776} C_VEL
LIN {X 0,Y 362.177,Z 890.179,A -85,B 0,C 180,E1 -13231.112,E2 -13231.112} C_VEL
LIN {X 0,Y 362.256,Z 890.175,A -85,B 0,C 180,E1 -13232.224,E2 -13232.224} C_VEL
LIN {X 0,Y 362.123,Z 890.189,A -85,B 0,C 180,E1 -13236.687,E2 -13236.687} C_VEL
LIN {X 0,Y 361.998,Z 890.204,A -85,B 0,C 180,E1 -13240.063,E2 -13240.063} C_VEL
LIN {X 0,Y 361.985,Z 890.204,A -85,B 0,C 180,E1 -13243.887,E2 -13243.887} C_VEL
LIN {X 0,Y 361.89,Z 890.216,A -85,B 0,C 180,E1 -13248.103,E2 -13248.103} C_VEL
LIN {X 0,Y 361.857,Z 890.22,A -85,B 0,C 180,E1 -13251.655,E2 -13251.655} C_VEL
LIN {X 0,Y 361.863,Z 890.223,A -85,B 0,C 180,E1 -13255.295,E2 -13255.295} C_VEL
LIN {X 0,Y 361.86,Z 890.223,A -85,B 0,C 180,E1 -13259.074,E2 -13259.074} C_VEL
LIN {X 0,Y 361.851,Z 890.221,A -85,B 0,C 180,E1 -13262.945,E2 -13262.945} C_VEL
LIN {X 0,Y 361.867,Z 890.224,A -85,B 0,C 180,E1 -13265.637,E2 -13265.637} C_VEL
LIN {X 0,Y 361.829,Z 890.223,A -85,B 0,C 180,E1 -13268.953,E2 -13268.953} C_VEL
LIN {X 0,Y 361.158,Z 890.312,A -85,B 0,C 180,E1 -13269.882,E2 -13269.882} C_VEL
LIN {X 0,Y 358.281,Z 890.667,A -85,B 0,C 180,E1 -13271.392,E2 -13271.392} C_VEL
LIN {X 0,Y 355.857,Z 890.967,A -85,B 0,C 180,E1 -13272.615,E2 -13272.615} C_VEL
LIN {X 0,Y 354.837,Z 891.096,A -85,B 0,C 180,E1 -13273.56,E2 -13273.56} C_VEL
LIN {X 0,Y 354.766,Z 891.108,A -85,B 0,C 180,E1 -13273.881,E2 -13273.881} C_VEL
LIN {X 0,Y 354.785,Z 891.102,A -85,B 0,C 180,E1 -13277.66,E2 -13277.66} C_VEL
LIN {X 0,Y 354.789,Z 891.102,A -85,B 0,C 180,E1 -13280.662,E2 -13280.662} C_VEL
LIN {X 0,Y 354.822,Z 891.101,A -85,B 0,C 180,E1 -13284.301,E2 -13284.301} C_VEL
LIN {X 0,Y 354.79,Z 891.099,A -85,B 0,C 180,E1 -13287.666,E2 -13287.666} C_VEL
LIN {X 0,Y 354.8,Z 891.098,A -85,B 0,C 180,E1 -13291.614,E2 -13291.614} C_VEL
LIN {X 0,Y 354.807,Z 891.099,A -85,B 0,C 180,E1 -13295.419,E2 -13295.419} C_VEL
LIN {X 0,Y 354.822,Z 891.102,A -85,B 0,C 180,E1 -13299.112,E2 -13299.112} C_VEL
LIN {X 0,Y 354.853,Z 891.093,A -85,B 0,C 180,E1 -13302.717,E2 -13302.717} C_VEL
LIN {X 0,Y 354.943,Z 891.08,A -85,B 0,C 180,E1 -13306.254,E2 -13306.254} C_VEL
LIN {X 0,Y 354.952,Z 891.084,A -85,B 0,C 180,E1 -13309.735,E2 -13309.735} C_VEL
LIN {X 0,Y 355.088,Z 891.064,A -85,B 0,C 180,E1 -13313.179,E2 -13313.179} C_VEL
LIN {X 0,Y 355.216,Z 891.051,A -85,B 0,C 180,E1 -13317.732,E2 -13317.732} C_VEL
LIN {X 0,Y 355.146,Z 891.055,A -85,B 0,C 180,E1 -13321.133,E2 -13321.133} C_VEL
LIN {X 0,Y 355.215,Z 891.051,A -85,B 0,C 180,E1 -13322.267,E2 -13322.267} C_VEL
LIN {X 0,Y 355.087,Z 891.064,A -85,B 0,C 180,E1 -13326.82,E2 -13326.82} C_VEL
LIN {X 0,Y 354.951,Z 891.084,A -85,B 0,C 180,E1 -13330.264,E2 -13330.264} C_VEL
LIN {X 0,Y 354.92,Z 891.084,A -85,B 0,C 180,E1 -13334.002,E2 -13334.002} C_VEL
LIN {X 0,Y 354.844,Z 891.093,A -85,B 0,C 180,E1 -13338.068,E2 -13338.068} C_VEL
LIN {X 0,Y 354.806,Z 891.097,A -85,B 0,C 180,E1 -13342.107,E2 -13342.107} C_VEL
LIN {X 0,Y 354.798,Z 891.099,A -85,B 0,C 180,E1 -13345.835,E2 -13345.835} C_VEL
LIN {X 0,Y 354.793,Z 891.102,A -85,B 0,C 180,E1 -13349.684,E2 -13349.684} C_VEL
LIN {X 0,Y 354.786,Z 891.1,A -85,B 0,C 180,E1 -13352.333,E2 -13352.333} C_VEL
LIN {X 0,Y 354.818,Z 891.102,A -85,B 0,C 180,E1 -13355.698,E2 -13355.698} C_VEL
LIN {X 0,Y 354.768,Z 891.105,A -85,B 0,C 180,E1 -13359.412,E2 -13359.412} C_VEL
LIN {X 0,Y 354.78,Z 891.1,A -85,B 0,C 180,E1 -13362.865,E2 -13362.865} C_VEL
LIN {X 0,Y 354.762,Z 891.109,A -85,B 0,C 180,E1 -13366.102,E2 -13366.102} C_VEL
LIN {X 0,Y 354.762,Z 891.103,A -85,B 0,C 180,E1 -13369.175,E2 -13369.175} C_VEL
LIN {X 0,Y 354.797,Z 891.105,A -85,B 0,C 180,E1 -13372.404,E2 -13372.404} C_VEL
LIN {X 0,Y 354.807,Z 891.099,A -85,B 0,C 180,E1 -13374.94,E2 -13374.94} C_VEL
LIN {X 0,Y 354.792,Z 891.104,A -85,B 0,C 180,E1 -13378.405,E2 -13378.405} C_VEL
LIN {X 0,Y 354.801,Z 891.098,A -85,B 0,C 180,E1 -13381.614,E2 -13381.614} C_VEL
LIN {X 0,Y 354.863,Z 891.254,A -85,B 0,C 180,E1 -13383.026,E2 -13383.026} C_VEL
LIN {X 0,Y 356.889,Z 902.245,A -85,B 0,C 180,E1 -13386.19,E2 -13386.19} C_VEL
LIN {X 0,Y 357.03,Z 905.52,A -85,B 0,C 180,E1 -13387.096,E2 -13387.096} C_VEL
LIN {X 0,Y 355.987,Z 917.791,A -85,B 0,C 180,E1 -13390.39,E2 -13390.39} C_VEL
LIN {X 0,Y 355.194,Z 927.948,A -85,B 0,C 180,E1 -13393.081,E2 -13393.081} C_VEL
LIN {X 0,Y 358.273,Z 955.785,A -85,B 0,C 180,E1 -13393.929,E2 -13393.929} C_VEL
LIN {X 0,Y 357.349,Z 1006.36,A -85,B 0,C 180,E1 -13395.259,E2 -13395.259} C_VEL
LIN {X 0,Y 356.781,Z 1017.789,A -85,B 0,C 180,E1 -13395.745,E2 -13395.745} C_VEL
LIN {X 0,Y 356.365,Z 1028.778,A -85,B 0,C 180,E1 -13396.456,E2 -13396.456} C_VEL
LIN {X 0,Y 355.867,Z 1037.25,A -85,B 0,C 180,E1 -13397.163,E2 -13397.163} C_VEL
LIN {X 0,Y 355.364,Z 1045.475,A -85,B 0,C 180,E1 -13398.015,E2 -13398.015} C_VEL
LIN {X 0,Y 354.944,Z 1052.301,A -85,B 0,C 180,E1 -13398.869,E2 -13398.869} C_VEL
LIN {X 0,Y 354.397,Z 1059.851,A -85,B 0,C 180,E1 -13400.007,E2 -13400.007} C_VEL
LIN {X 0,Y 353.952,Z 1067.525,A -85,B 0,C 180,E1 -13401.435,E2 -13401.435} C_VEL
LIN {X 0,Y 353.701,Z 1073.498,A -85,B 0,C 180,E1 -13402.866,E2 -13402.866} C_VEL
LIN {X 0,Y 353.415,Z 1078.174,A -85,B 0,C 180,E1 -13404.293,E2 -13404.293} C_VEL
LIN {X 0,Y 353.431,Z 1081.187,A -85,B 0,C 180,E1 -13405.438,E2 -13405.438} C_VEL
LIN {X 0,Y 353.28,Z 1083.535,A -85,B 0,C 180,E1 -13406.578,E2 -13406.578} C_VEL
LIN {X 0,Y 353.266,Z 1085.227,A -85,B 0,C 180,E1 -13407.719,E2 -13407.719} C_VEL
LIN {X 0,Y 353.372,Z 1086.337,A -85,B 0,C 180,E1 -13408.86,E2 -13408.86} C_VEL
LIN {X 0,Y 353.375,Z 1086.91,A -85,B 0,C 180,E1 -13410,E2 -13410} C_VEL
LIN {X 0,Y 353.286,Z 1086.958,A -85,B 0,C 180,E1 -13411.14,E2 -13411.14} C_VEL
LIN {X 0,Y 353.22,Z 1086.482,A -85,B 0,C 180,E1 -13412.28,E2 -13412.28} C_VEL
LIN {X 0,Y 353.271,Z 1085.392,A -85,B 0,C 180,E1 -13413.421,E2 -13413.421} C_VEL
LIN {X 0,Y 353.386,Z 1082.752,A -85,B 0,C 180,E1 -13415.134,E2 -13415.134} C_VEL
LIN {X 0,Y 353.605,Z 1078.694,A -85,B 0,C 180,E1 -13416.849,E2 -13416.849} C_VEL
LIN {X 0,Y 354.026,Z 1073.177,A -85,B 0,C 180,E1 -13418.562,E2 -13418.562} C_VEL
LIN {X 0,Y 354.619,Z 1067.277,A -85,B 0,C 180,E1 -13419.986,E2 -13419.986} C_VEL
LIN {X 0,Y 355.341,Z 1059.856,A -85,B 0,C 180,E1 -13421.407,E2 -13421.407} C_VEL
LIN {X 0,Y 356.178,Z 1051.489,A -85,B 0,C 180,E1 -13422.68,E2 -13422.68} C_VEL
LIN {X 0,Y 356.889,Z 1043.556,A -85,B 0,C 180,E1 -13423.669,E2 -13423.669} C_VEL
LIN {X 0,Y 357.763,Z 1033.794,A -85,B 0,C 180,E1 -13424.65,E2 -13424.65} C_VEL
LIN {X 0,Y 358.715,Z 1022.841,A -85,B 0,C 180,E1 -13425.482,E2 -13425.482} C_VEL
LIN {X 0,Y 359.547,Z 1012.261,A -85,B 0,C 180,E1 -13426.064,E2 -13426.064} C_VEL
LIN {X 0,Y 360.05,Z 1001.707,A -85,B 0,C 180,E1 -13426.478,E2 -13426.478} C_VEL
LIN {X 0,Y 361.495,Z 956.085,A -85,B 0,C 180,E1 -13427.793,E2 -13427.793} C_VEL
LIN {X 0,Y 360.033,Z 942.551,A -85,B 0,C 180,E1 -13428.346,E2 -13428.346} C_VEL
LIN {X 0,Y 357.206,Z 928.204,A -85,B 0,C 180,E1 -13429.068,E2 -13429.068} C_VEL
LIN {X 0,Y 356.537,Z 925.096,A -85,B 0,C 180,E1 -13429.258,E2 -13429.258} C_VEL
LIN {X 0,Y 358.195,Z 911.94,A -85,B 0,C 180,E1 -13433.105,E2 -13433.105} C_VEL
LIN {X 0,Y 358.276,Z 908.077,A -85,B 0,C 180,E1 -13434.327,E2 -13434.327} C_VEL
LIN {X 0,Y 357.034,Z 900.811,A -85,B 0,C 180,E1 -13436.92,E2 -13436.92} C_VEL
LIN {X 0,Y 355.502,Z 894.051,A -85,B 0,C 180,E1 -13439.619,E2 -13439.619} C_VEL
LIN {X 0,Y 354.789,Z 891.106,A -85,B 0,C 180,E1 -13440.999,E2 -13440.999} C_VEL
LIN {X 0,Y 354.804,Z 891.105,A -85,B 0,C 180,E1 -13443.702,E2 -13443.702} C_VEL
LIN {X 0,Y 354.789,Z 891.103,A -85,B 0,C 180,E1 -13446.46,E2 -13446.46} C_VEL
LIN {X 0,Y 354.766,Z 891.107,A -85,B 0,C 180,E1 -13449.413,E2 -13449.413} C_VEL
LIN {X 0,Y 354.778,Z 891.105,A -85,B 0,C 180,E1 -13452.866,E2 -13452.866} C_VEL
LIN {X 0,Y 354.76,Z 891.109,A -85,B 0,C 180,E1 -13456.103,E2 -13456.103} C_VEL
LIN {X 0,Y 354.76,Z 891.106,A -85,B 0,C 180,E1 -13459.176,E2 -13459.176} C_VEL
LIN {X 0,Y 354.795,Z 891.103,A -85,B 0,C 180,E1 -13462.405,E2 -13462.405} C_VEL
LIN {X 0,Y 354.805,Z 891.101,A -85,B 0,C 180,E1 -13464.941,E2 -13464.941} C_VEL
LIN {X 0,Y 354.791,Z 891.104,A -85,B 0,C 180,E1 -13468.406,E2 -13468.406} C_VEL
LIN {X 0,Y 354.786,Z 891.104,A -85,B 0,C 180,E1 -13471.614,E2 -13471.614} C_VEL
LIN {X 0,Y 354.818,Z 891.119,A -85,B 0,C 180,E1 -13475.109,E2 -13475.109} C_VEL
LIN {X 0,Y 356.104,Z 897.107,A -85,B 0,C 180,E1 -13478.061,E2 -13478.061} C_VEL
LIN {X 0,Y 357.116,Z 903.413,A -85,B 0,C 180,E1 -13480.845,E2 -13480.845} C_VEL
LIN {X 0,Y 357.365,Z 904.369,A -85,B 0,C 180,E1 -13480.946,E2 -13480.946} C_VEL
LIN {X 0,Y 360.491,Z 914.088,A -85,B 0,C 180,E1 -13481.568,E2 -13481.568} C_VEL
LIN {X 0,Y 362.413,Z 923.254,A -85,B 0,C 180,E1 -13482.03,E2 -13482.03} C_VEL
LIN {X 0,Y 360.222,Z 980.71,A -85,B 0,C 180,E1 -13483.713,E2 -13483.713} C_VEL
LIN {X 0,Y 359.627,Z 993.352,A -85,B 0,C 180,E1 -13484.34,E2 -13484.34} C_VEL
LIN {X 0,Y 358.955,Z 1002.523,A -85,B 0,C 180,E1 -13484.965,E2 -13484.965} C_VEL
LIN {X 0,Y 358.258,Z 1012.05,A -85,B 0,C 180,E1 -13485.806,E2 -13485.806} C_VEL
LIN {X 0,Y 357.384,Z 1022.065,A -85,B 0,C 180,E1 -13486.93,E2 -13486.93} C_VEL
LIN {X 0,Y 356.625,Z 1029.893,A -85,B 0,C 180,E1 -13488.058,E2 -13488.058} C_VEL
LIN {X 0,Y 355.918,Z 1036.351,A -85,B 0,C 180,E1 -13489.188,E2 -13489.188} C_VEL
LIN {X 0,Y 355.28,Z 1041.729,A -85,B 0,C 180,E1 -13490.321,E2 -13490.321} C_VEL
LIN {X 0,Y 354.824,Z 1046.201,A -85,B 0,C 180,E1 -13491.457,E2 -13491.457} C_VEL
LIN {X 0,Y 354.388,Z 1050.799,A -85,B 0,C 180,E1 -13492.919,E2 -13492.919} C_VEL
LIN {X 0,Y 353.868,Z 1054.159,A -85,B 0,C 180,E1 -13494.301,E2 -13494.301} C_VEL
LIN {X 0,Y 353.664,Z 1056.245,A -85,B 0,C 180,E1 -13495.441,E2 -13495.441} C_VEL
LIN {X 0,Y 353.618,Z 1057.776,A -85,B 0,C 180,E1 -13496.582,E2 -13496.582} C_VEL
LIN {X 0,Y 353.519,Z 1058.717,A -85,B 0,C 180,E1 -13497.722,E2 -13497.722} C_VEL
LIN {X 0,Y 353.396,Z 1059.069,A -85,B 0,C 180,E1 -13498.861,E2 -13498.861} C_VEL
LIN {X 0,Y 353.329,Z 1058.908,A -85,B 0,C 180,E1 -13500.001,E2 -13500.001} C_VEL
LIN {X 0,Y 353.303,Z 1058.236,A -85,B 0,C 180,E1 -13501.14,E2 -13501.14} C_VEL
LIN {X 0,Y 353.322,Z 1057.047,A -85,B 0,C 180,E1 -13502.281,E2 -13502.281} C_VEL
LIN {X 0,Y 353.444,Z 1054.084,A -85,B 0,C 180,E1 -13503.991,E2 -13503.991} C_VEL
LIN {X 0,Y 353.635,Z 1049.792,A -85,B 0,C 180,E1 -13505.703,E2 -13505.703} C_VEL
LIN {X 0,Y 354.004,Z 1043.978,A -85,B 0,C 180,E1 -13507.415,E2 -13507.415} C_VEL
LIN {X 0,Y 354.299,Z 1037.568,A -85,B 0,C 180,E1 -13508.844,E2 -13508.844} C_VEL
LIN {X 0,Y 354.763,Z 1031.304,A -85,B 0,C 180,E1 -13509.983,E2 -13509.983} C_VEL
LIN {X 0,Y 355.223,Z 1023.691,A -85,B 0,C 180,E1 -13511.123,E2 -13511.123} C_VEL
LIN {X 0,Y 355.683,Z 1016.832,A -85,B 0,C 180,E1 -13511.975,E2 -13511.975} C_VEL
LIN {X 0,Y 356.111,Z 1008.548,A -85,B 0,C 180,E1 -13512.828,E2 -13512.828} C_VEL
LIN {X 0,Y 356.64,Z 998.164,A -85,B 0,C 180,E1 -13513.679,E2 -13513.679} C_VEL
LIN {X 0,Y 357.036,Z 986.737,A -85,B 0,C 180,E1 -13514.354,E2 -13514.354} C_VEL
LIN {X 0,Y 357.357,Z 977.325,A -85,B 0,C 180,E1 -13514.741,E2 -13514.741} C_VEL
LIN {X 0,Y 358.394,Z 919.894,A -85,B 0,C 180,E1 -13516.241,E2 -13516.241} C_VEL
LIN {X 0,Y 355.278,Z 900.088,A -85,B 0,C 180,E1 -13516.891,E2 -13516.891} C_VEL
LIN {X 0,Y 355.411,Z 895.372,A -85,B 0,C 180,E1 -13518.445,E2 -13518.445} C_VEL
LIN {X 0,Y 354.929,Z 891.083,A -85,B 0,C 180,E1 -13519.973,E2 -13519.973} C_VEL
LIN {X 0,Y 354.806,Z 891.098,A -85,B 0,C 180,E1 -13524.333,E2 -13524.333} C_VEL
LIN {X 0,Y 354.794,Z 891.104,A -85,B 0,C 180,E1 -13527.104,E2 -13527.104} C_VEL
LIN {X 0,Y 354.794,Z 891.102,A -85,B 0,C 180,E1 -13529.685,E2 -13529.685} C_VEL
LIN {X 0,Y 354.788,Z 891.1,A -85,B 0,C 180,E1 -13532.334,E2 -13532.334} C_VEL
LIN {X 0,Y 354.82,Z 891.101,A -85,B 0,C 180,E1 -13535.699,E2 -13535.699} C_VEL
LIN {X 0,Y 354.77,Z 891.105,A -85,B 0,C 180,E1 -13539.413,E2 -13539.413} C_VEL
LIN {X 0,Y 354.783,Z 891.1,A -85,B 0,C 180,E1 -13542.866,E2 -13542.866} C_VEL
LIN {X 0,Y 354.765,Z 891.109,A -85,B 0,C 180,E1 -13546.103,E2 -13546.103} C_VEL
LIN {X 0,Y 354.765,Z 891.102,A -85,B 0,C 180,E1 -13549.176,E2 -13549.176} C_VEL
LIN {X 0,Y 354.801,Z 891.104,A -85,B 0,C 180,E1 -13552.405,E2 -13552.405} C_VEL
LIN {X 0,Y 354.811,Z 891.099,A -85,B 0,C 180,E1 -13554.941,E2 -13554.941} C_VEL
LIN {X 0,Y 354.796,Z 891.103,A -85,B 0,C 180,E1 -13558.406,E2 -13558.406} C_VEL
LIN {X 0,Y 354.799,Z 891.098,A -85,B 0,C 180,E1 -13561.615,E2 -13561.615} C_VEL
LIN {X 0,Y 354.838,Z 891.094,A -85,B 0,C 180,E1 -13565.658,E2 -13565.658} C_VEL
LIN {X 0,Y 354.823,Z 891.102,A -85,B 0,C 180,E1 -13569.113,E2 -13569.113} C_VEL
LIN {X 0,Y 354.867,Z 891.091,A -85,B 0,C 180,E1 -13572.719,E2 -13572.719} C_VEL
LIN {X 0,Y 354.954,Z 891.079,A -85,B 0,C 180,E1 -13576.255,E2 -13576.255} C_VEL
LIN {X 0,Y 354.954,Z 891.084,A -85,B 0,C 180,E1 -13579.735,E2 -13579.735} C_VEL
LIN {X 0,Y 355.089,Z 891.064,A -85,B 0,C 180,E1 -13583.18,E2 -13583.18} C_VEL
LIN {X 0,Y 355.218,Z 891.051,A -85,B 0,C 180,E1 -13587.732,E2 -13587.732} C_VEL
LIN {X 0,Y 355.149,Z 891.055,A -85,B 0,C 180,E1 -13591.134,E2 -13591.134} C_VEL
LIN {X 0,Y 355.218,Z 891.051,A -85,B 0,C 180,E1 -13592.268,E2 -13592.268} C_VEL
LIN {X 0,Y 355.089,Z 891.064,A -85,B 0,C 180,E1 -13596.82,E2 -13596.82} C_VEL
LIN {X 0,Y 354.954,Z 891.083,A -85,B 0,C 180,E1 -13600.265,E2 -13600.265} C_VEL
LIN {X 0,Y 354.923,Z 891.084,A -85,B 0,C 180,E1 -13604.003,E2 -13604.003} C_VEL
LIN {X 0,Y 354.847,Z 891.093,A -85,B 0,C 180,E1 -13608.068,E2 -13608.068} C_VEL
LIN {X 0,Y 354.809,Z 891.097,A -85,B 0,C 180,E1 -13612.108,E2 -13612.108} C_VEL
LIN {X 0,Y 354.802,Z 891.099,A -85,B 0,C 180,E1 -13615.835,E2 -13615.835} C_VEL
LIN {X 0,Y 354.797,Z 891.101,A -85,B 0,C 180,E1 -13619.684,E2 -13619.684} C_VEL
LIN {X 0,Y 354.79,Z 891.099,A -85,B 0,C 180,E1 -13622.333,E2 -13622.333} C_VEL
LIN {X 0,Y 354.822,Z 891.101,A -85,B 0,C 180,E1 -13625.698,E2 -13625.698} C_VEL
LIN {X 0,Y 354.772,Z 891.105,A -85,B 0,C 180,E1 -13629.412,E2 -13629.412} C_VEL
LIN {X 0,Y 354.785,Z 891.1,A -85,B 0,C 180,E1 -13632.866,E2 -13632.866} C_VEL
LIN {X 0,Y 354.766,Z 891.108,A -85,B 0,C 180,E1 -13633.881,E2 -13633.881} C_VEL
LIN {X 0,Y 354.132,Z 891.195,A -85,B 0,C 180,E1 -13634.828,E2 -13634.828} C_VEL
LIN {X 0,Y 351.298,Z 891.549,A -85,B 0,C 180,E1 -13636.368,E2 -13636.368} C_VEL
LIN {X 0,Y 348.864,Z 891.845,A -85,B 0,C 180,E1 -13637.614,E2 -13637.614} C_VEL
LIN {X 0,Y 347.8,Z 891.973,A -85,B 0,C 180,E1 -13638.579,E2 -13638.579} C_VEL
LIN {X 0,Y 347.704,Z 891.982,A -85,B 0,C 180,E1 -13638.905,E2 -13638.905} C_VEL
LIN {X 0,Y 347.758,Z 891.978,A -85,B 0,C 180,E1 -13642.678,E2 -13642.678} C_VEL
LIN {X 0,Y 347.752,Z 891.978,A -85,B 0,C 180,E1 -13645.956,E2 -13645.956} C_VEL
LIN {X 0,Y 347.739,Z 891.978,A -85,B 0,C 180,E1 -13649.65,E2 -13649.65} C_VEL
LIN {X 0,Y 347.737,Z 891.978,A -85,B 0,C 180,E1 -13653.599,E2 -13653.599} C_VEL
LIN {X 0,Y 347.751,Z 891.976,A -85,B 0,C 180,E1 -13656.158,E2 -13656.158} C_VEL
LIN {X 0,Y 347.77,Z 891.974,A -85,B 0,C 180,E1 -13659.906,E2 -13659.906} C_VEL
LIN {X 0,Y 347.796,Z 891.974,A -85,B 0,C 180,E1 -13663.566,E2 -13663.566} C_VEL
LIN {X 0,Y 347.886,Z 891.963,A -85,B 0,C 180,E1 -13667.16,E2 -13667.16} C_VEL
LIN {X 0,Y 347.936,Z 891.953,A -85,B 0,C 180,E1 -13670.7,E2 -13670.7} C_VEL
LIN {X 0,Y 348.038,Z 891.943,A -85,B 0,C 180,E1 -13674.205,E2 -13674.205} C_VEL
LIN {X 0,Y 348.153,Z 891.93,A -85,B 0,C 180,E1 -13677.686,E2 -13677.686} C_VEL
LIN {X 0,Y 348.118,Z 891.93,A -85,B 0,C 180,E1 -13681.156,E2 -13681.156} C_VEL
LIN {X 0,Y 348.153,Z 891.931,A -85,B 0,C 180,E1 -13682.313,E2 -13682.313} C_VEL
LIN {X 0,Y 348.054,Z 891.939,A -85,B 0,C 180,E1 -13686.958,E2 -13686.958} C_VEL
LIN {X 0,Y 347.891,Z 891.965,A -85,B 0,C 180,E1 -13690.475,E2 -13690.475} C_VEL
LIN {X 0,Y 347.86,Z 891.964,A -85,B 0,C 180,E1 -13694.122,E2 -13694.122} C_VEL
LIN {X 0,Y 347.795,Z 891.972,A -85,B 0,C 180,E1 -13698.241,E2 -13698.241} C_VEL
LIN {X 0,Y 347.764,Z 891.975,A -85,B 0,C 180,E1 -13701.623,E2 -13701.623} C_VEL
LIN {X 0,Y 347.737,Z 891.984,A -85,B 0,C 180,E1 -13705.114,E2 -13705.114} C_VEL
LIN {X 0,Y 347.724,Z 891.981,A -85,B 0,C 180,E1 -13707.701,E2 -13707.701} C_VEL
LIN {X 0,Y 347.736,Z 891.978,A -85,B 0,C 180,E1 -13710.349,E2 -13710.349} C_VEL
LIN {X 0,Y 347.748,Z 891.978,A -85,B 0,C 180,E1 -13714.043,E2 -13714.043} C_VEL
LIN {X 0,Y 347.754,Z 891.979,A -85,B 0,C 180,E1 -13717.321,E2 -13717.321} C_VEL
LIN {X 0,Y 347.695,Z 891.985,A -85,B 0,C 180,E1 -13720.302,E2 -13720.302} C_VEL
LIN {X 0,Y 347.72,Z 891.982,A -85,B 0,C 180,E1 -13723.408,E2 -13723.408} C_VEL
LIN {X 0,Y 347.722,Z 891.981,A -85,B 0,C 180,E1 -13726.686,E2 -13726.686} C_VEL
LIN {X 0,Y 347.7,Z 891.989,A -85,B 0,C 180,E1 -13730.182,E2 -13730.182} C_VEL
LIN {X 0,Y 347.753,Z 891.979,A -85,B 0,C 180,E1 -13732.678,E2 -13732.678} C_VEL
LIN {X 0,Y 347.747,Z 891.978,A -85,B 0,C 180,E1 -13735.956,E2 -13735.956} C_VEL
LIN {X 0,Y 347.735,Z 891.978,A -85,B 0,C 180,E1 -13739.65,E2 -13739.65} C_VEL
LIN {X 0,Y 347.81,Z 892.146,A -85,B 0,C 180,E1 -13742.888,E2 -13742.888} C_VEL
LIN {X 0,Y 349.956,Z 903.816,A -85,B 0,C 180,E1 -13746.318,E2 -13746.318} C_VEL
LIN {X 0,Y 349.709,Z 909.394,A -85,B 0,C 180,E1 -13747.863,E2 -13747.863} C_VEL
LIN {X 0,Y 348.603,Z 922.184,A -85,B 0,C 180,E1 -13751.358,E2 -13751.358} C_VEL
LIN {X 0,Y 348.183,Z 927.61,A -85,B 0,C 180,E1 -13752.83,E2 -13752.83} C_VEL
LIN {X 0,Y 351.282,Z 957.038,A -85,B 0,C 180,E1 -13753.764,E2 -13753.764} C_VEL
LIN {X 0,Y 350.325,Z 1006.467,A -85,B 0,C 180,E1 -13755.105,E2 -13755.105} C_VEL
LIN {X 0,Y 349.746,Z 1017.718,A -85,B 0,C 180,E1 -13755.601,E2 -13755.601} C_VEL
LIN {X 0,Y 349.331,Z 1028.635,A -85,B 0,C 180,E1 -13756.326,E2 -13756.326} C_VEL
LIN {X 0,Y 348.811,Z 1037.075,A -85,B 0,C 180,E1 -13757.047,E2 -13757.047} C_VEL
LIN {X 0,Y 348.309,Z 1045.287,A -85,B 0,C 180,E1 -13757.916,E2 -13757.916} C_VEL
LIN {X 0,Y 347.876,Z 1052.102,A -85,B 0,C 180,E1 -13758.787,E2 -13758.787} C_VEL
LIN {X 0,Y 347.38,Z 1058.77,A -85,B 0,C 180,E1 -13759.803,E2 -13759.803} C_VEL
LIN {X 0,Y 346.998,Z 1065.122,A -85,B 0,C 180,E1 -13760.969,E2 -13760.969} C_VEL
LIN {X 0,Y 346.66,Z 1071.594,A -85,B 0,C 180,E1 -13762.427,E2 -13762.427} C_VEL
LIN {X 0,Y 346.338,Z 1077.519,A -85,B 0,C 180,E1 -13764.176,E2 -13764.176} C_VEL
LIN {X 0,Y 346.342,Z 1080.61,A -85,B 0,C 180,E1 -13765.344,E2 -13765.344} C_VEL
LIN {X 0,Y 346.208,Z 1082.992,A -85,B 0,C 180,E1 -13766.508,E2 -13766.508} C_VEL
LIN {X 0,Y 346.176,Z 1084.728,A -85,B 0,C 180,E1 -13767.673,E2 -13767.673} C_VEL
LIN {X 0,Y 346.277,Z 1085.915,A -85,B 0,C 180,E1 -13768.837,E2 -13768.837} C_VEL
LIN {X 0,Y 346.296,Z 1086.565,A -85,B 0,C 180,E1 -13770,E2 -13770} C_VEL
LIN {X 0,Y 346.187,Z 1086.689,A -85,B 0,C 180,E1 -13771.163,E2 -13771.163} C_VEL
LIN {X 0,Y 346.129,Z 1086.249,A -85,B 0,C 180,E1 -13772.327,E2 -13772.327} C_VEL
LIN {X 0,Y 346.196,Z 1085.19,A -85,B 0,C 180,E1 -13773.491,E2 -13773.491} C_VEL
LIN {X 0,Y 346.289,Z 1082.66,A -85,B 0,C 180,E1 -13775.24,E2 -13775.24} C_VEL
LIN {X 0,Y 346.545,Z 1078.687,A -85,B 0,C 180,E1 -13776.989,E2 -13776.989} C_VEL
LIN {X 0,Y 346.923,Z 1074.295,A -85,B 0,C 180,E1 -13778.445,E2 -13778.445} C_VEL
LIN {X 0,Y 347.475,Z 1068.74,A -85,B 0,C 180,E1 -13779.899,E2 -13779.899} C_VEL
LIN {X 0,Y 348.059,Z 1063.31,A -85,B 0,C 180,E1 -13781.059,E2 -13781.059} C_VEL
LIN {X 0,Y 348.776,Z 1056.798,A -85,B 0,C 180,E1 -13782.215,E2 -13782.215} C_VEL
LIN {X 0,Y 349.607,Z 1048.935,A -85,B 0,C 180,E1 -13783.366,E2 -13783.366} C_VEL
LIN {X 0,Y 350.597,Z 1039.198,A -85,B 0,C 180,E1 -13784.511,E2 -13784.511} C_VEL
LIN {X 0,Y 351.424,Z 1029.947,A -85,B 0,C 180,E1 -13785.366,E2 -13785.366} C_VEL
LIN {X 0,Y 352.239,Z 1021.278,A -85,B 0,C 180,E1 -13785.997,E2 -13785.997} C_VEL
LIN {X 0,Y 353.048,Z 1011.235,A -85,B 0,C 180,E1 -13786.554,E2 -13786.554} C_VEL
LIN {X 0,Y 353.667,Z 999.656,A -85,B 0,C 180,E1 -13787.007,E2 -13787.007} C_VEL
LIN {X 0,Y 355.113,Z 957.245,A -85,B 0,C 180,E1 -13788.256,E2 -13788.256} C_VEL
LIN {X 0,Y 353.748,Z 943.797,A -85,B 0,C 180,E1 -13788.835,E2 -13788.835} C_VEL
LIN {X 0,Y 350.965,Z 929.844,A -85,B 0,C 180,E1 -13789.581,E2 -13789.581} C_VEL
LIN {X 0,Y 349.809,Z 924.663,A -85,B 0,C 180,E1 -13789.909,E2 -13789.909} C_VEL
LIN {X 0,Y 351.25,Z 914.319,A -85,B 0,C 180,E1 -13793.017,E2 -13793.017} C_VEL
LIN {X 0,Y 351.492,Z 910.655,A -85,B 0,C 180,E1 -13794.198,E2 -13794.198} C_VEL
LIN {X 0,Y 350.749,Z 905.182,A -85,B 0,C 180,E1 -13796.156,E2 -13796.156} C_VEL
LIN {X 0,Y 349.278,Z 898.355,A -85,B 0,C 180,E1 -13798.876,E2 -13798.876} C_VEL
LIN {X 0,Y 347.744,Z 891.984,A -85,B 0,C 180,E1 -13801.81,E2 -13801.81} C_VEL
LIN {X 0,Y 347.781,Z 891.979,A -85,B 0,C 180,E1 -13805.876,E2 -13805.876} C_VEL
LIN {X 0,Y 347.728,Z 891.984,A -85,B 0,C 180,E1 -13808.796,E2 -13808.796} C_VEL
LIN {X 0,Y 347.737,Z 891.982,A -85,B 0,C 180,E1 -13811.832,E2 -13811.832} C_VEL
LIN {X 0,Y 347.698,Z 891.987,A -85,B 0,C 180,E1 -13815.028,E2 -13815.028} C_VEL
LIN {X 0,Y 347.735,Z 891.981,A -85,B 0,C 180,E1 -13818.4,E2 -13818.4} C_VEL
LIN {X 0,Y 347.759,Z 891.979,A -85,B 0,C 180,E1 -13822.014,E2 -13822.014} C_VEL
LIN {X 0,Y 347.741,Z 891.981,A -85,B 0,C 180,E1 -13825.536,E2 -13825.536} C_VEL
LIN {X 0,Y 347.742,Z 891.982,A -85,B 0,C 180,E1 -13828.301,E2 -13828.301} C_VEL
LIN {X 0,Y 347.739,Z 891.984,A -85,B 0,C 180,E1 -13830.984,E2 -13830.984} C_VEL
LIN {X 0,Y 347.786,Z 892.087,A -85,B 0,C 180,E1 -13834.329,E2 -13834.329} C_VEL
LIN {X 0,Y 349.136,Z 898.198,A -85,B 0,C 180,E1 -13837.514,E2 -13837.514} C_VEL
LIN {X 0,Y 350.142,Z 904.046,A -85,B 0,C 180,E1 -13840.224,E2 -13840.224} C_VEL
LIN {X 0,Y 353.457,Z 912.881,A -85,B 0,C 180,E1 -13840.879,E2 -13840.879} C_VEL
LIN {X 0,Y 356.112,Z 923.722,A -85,B 0,C 180,E1 -13841.507,E2 -13841.507} C_VEL
LIN {X 0,Y 353.758,Z 981.308,A -85,B 0,C 180,E1 -13843.258,E2 -13843.258} C_VEL
LIN {X 0,Y 353.221,Z 992.722,A -85,B 0,C 180,E1 -13843.826,E2 -13843.826} C_VEL
LIN {X 0,Y 352.412,Z 1002.887,A -85,B 0,C 180,E1 -13844.531,E2 -13844.531} C_VEL
LIN {X 0,Y 351.644,Z 1012.332,A -85,B 0,C 180,E1 -13845.385,E2 -13845.385} C_VEL
LIN {X 0,Y 350.696,Z 1022.302,A -85,B 0,C 180,E1 -13846.529,E2 -13846.529} C_VEL
LIN {X 0,Y 349.773,Z 1030.993,A -85,B 0,C 180,E1 -13847.821,E2 -13847.821} C_VEL
LIN {X 0,Y 349.022,Z 1037.34,A -85,B 0,C 180,E1 -13848.972,E2 -13848.972} C_VEL
LIN {X 0,Y 348.345,Z 1042.617,A -85,B 0,C 180,E1 -13850.126,E2 -13850.126} C_VEL
LIN {X 0,Y 347.864,Z 1046.998,A -85,B 0,C 180,E1 -13851.285,E2 -13851.285} C_VEL
LIN {X 0,Y 347.434,Z 1051.121,A -85,B 0,C 180,E1 -13852.637,E2 -13852.637} C_VEL
LIN {X 0,Y 346.841,Z 1054.749,A -85,B 0,C 180,E1 -13854.186,E2 -13854.186} C_VEL
LIN {X 0,Y 346.601,Z 1056.748,A -85,B 0,C 180,E1 -13855.348,E2 -13855.348} C_VEL
LIN {X 0,Y 346.536,Z 1058.202,A -85,B 0,C 180,E1 -13856.512,E2 -13856.512} C_VEL
LIN {X 0,Y 346.434,Z 1059.118,A -85,B 0,C 180,E1 -13857.675,E2 -13857.675} C_VEL
LIN {X 0,Y 346.306,Z 1059.416,A -85,B 0,C 180,E1 -13858.838,E2 -13858.838} C_VEL
LIN {X 0,Y 346.234,Z 1059.174,A -85,B 0,C 180,E1 -13860.001,E2 -13860.001} C_VEL
LIN {X 0,Y 346.206,Z 1058.422,A -85,B 0,C 180,E1 -13861.164,E2 -13861.164} C_VEL
LIN {X 0,Y 346.227,Z 1057.143,A -85,B 0,C 180,E1 -13862.327,E2 -13862.327} C_VEL
LIN {X 0,Y 346.297,Z 1055.311,A -85,B 0,C 180,E1 -13863.491,E2 -13863.491} C_VEL
LIN {X 0,Y 346.514,Z 1051.302,A -85,B 0,C 180,E1 -13865.237,E2 -13865.237} C_VEL
LIN {X 0,Y 346.702,Z 1047.261,A -85,B 0,C 180,E1 -13866.574,E2 -13866.574} C_VEL
LIN {X 0,Y 346.993,Z 1042.43,A -85,B 0,C 180,E1 -13867.858,E2 -13867.858} C_VEL
LIN {X 0,Y 347.387,Z 1035.63,A -85,B 0,C 180,E1 -13869.315,E2 -13869.315} C_VEL
LIN {X 0,Y 347.993,Z 1027.109,A -85,B 0,C 180,E1 -13870.767,E2 -13870.767} C_VEL
LIN {X 0,Y 348.55,Z 1018.375,A -85,B 0,C 180,E1 -13871.928,E2 -13871.928} C_VEL
LIN {X 0,Y 349.023,Z 1010.375,A -85,B 0,C 180,E1 -13872.798,E2 -13872.798} C_VEL
LIN {X 0,Y 349.438,Z 1002.214,A -85,B 0,C 180,E1 -13873.522,E2 -13873.522} C_VEL
LIN {X 0,Y 349.874,Z 992.969,A -85,B 0,C 180,E1 -13874.171,E2 -13874.171} C_VEL
LIN {X 0,Y 350.165,Z 981.876,A -85,B 0,C 180,E1 -13874.753,E2 -13874.753} C_VEL
LIN {X 0,Y 350.664,Z 965.959,A -85,B 0,C 180,E1 -13875.244,E2 -13875.244} C_VEL
LIN {X 0,Y 351.425,Z 920.627,A -85,B 0,C 180,E1 -13876.441,E2 -13876.441} C_VEL
LIN {X 0,Y 348.276,Z 900.333,A -85,B 0,C 180,E1 -13877.127,E2 -13877.127} C_VEL
LIN {X 0,Y 348.306,Z 895.25,A -85,B 0,C 180,E1 -13878.836,E2 -13878.836} C_VEL
LIN {X 0,Y 347.889,Z 891.96,A -85,B 0,C 180,E1 -13880.01,E2 -13880.01} C_VEL
LIN {X 0,Y 347.772,Z 891.975,A -85,B 0,C 180,E1 -13884.579,E2 -13884.579} C_VEL
LIN {X 0,Y 347.725,Z 891.981,A -85,B 0,C 180,E1 -13887.702,E2 -13887.702} C_VEL
LIN {X 0,Y 347.737,Z 891.978,A -85,B 0,C 180,E1 -13890.35,E2 -13890.35} C_VEL
LIN {X 0,Y 347.75,Z 891.978,A -85,B 0,C 180,E1 -13894.044,E2 -13894.044} C_VEL
LIN {X 0,Y 347.756,Z 891.979,A -85,B 0,C 180,E1 -13897.322,E2 -13897.322} C_VEL
LIN {X 0,Y 347.697,Z 891.985,A -85,B 0,C 180,E1 -13900.303,E2 -13900.303} C_VEL
LIN {X 0,Y 347.723,Z 891.981,A -85,B 0,C 180,E1 -13903.409,E2 -13903.409} C_VEL
LIN {X 0,Y 347.725,Z 891.981,A -85,B 0,C 180,E1 -13906.687,E2 -13906.687} C_VEL
LIN {X 0,Y 347.703,Z 891.988,A -85,B 0,C 180,E1 -13910.183,E2 -13910.183} C_VEL
LIN {X 0,Y 347.757,Z 891.979,A -85,B 0,C 180,E1 -13912.679,E2 -13912.679} C_VEL
LIN {X 0,Y 347.751,Z 891.978,A -85,B 0,C 180,E1 -13915.957,E2 -13915.957} C_VEL
LIN {X 0,Y 347.739,Z 891.978,A -85,B 0,C 180,E1 -13919.651,E2 -13919.651} C_VEL
LIN {X 0,Y 347.741,Z 891.978,A -85,B 0,C 180,E1 -13923.601,E2 -13923.601} C_VEL
LIN {X 0,Y 347.765,Z 891.975,A -85,B 0,C 180,E1 -13926.16,E2 -13926.16} C_VEL
LIN {X 0,Y 347.772,Z 891.974,A -85,B 0,C 180,E1 -13929.907,E2 -13929.907} C_VEL
LIN {X 0,Y 347.824,Z 891.971,A -85,B 0,C 180,E1 -13933.568,E2 -13933.568} C_VEL
LIN {X 0,Y 347.89,Z 891.963,A -85,B 0,C 180,E1 -13937.161,E2 -13937.161} C_VEL
LIN {X 0,Y 347.937,Z 891.953,A -85,B 0,C 180,E1 -13940.701,E2 -13940.701} C_VEL
LIN {X 0,Y 348.039,Z 891.942,A -85,B 0,C 180,E1 -13944.205,E2 -13944.205} C_VEL
LIN {X 0,Y 348.156,Z 891.93,A -85,B 0,C 180,E1 -13947.686,E2 -13947.686} C_VEL
LIN {X 0,Y 348.12,Z 891.93,A -85,B 0,C 180,E1 -13951.157,E2 -13951.157} C_VEL
LIN {X 0,Y 348.155,Z 891.93,A -85,B 0,C 180,E1 -13952.314,E2 -13952.314} C_VEL
LIN {X 0,Y 348.057,Z 891.939,A -85,B 0,C 180,E1 -13956.959,E2 -13956.959} C_VEL
LIN {X 0,Y 347.894,Z 891.965,A -85,B 0,C 180,E1 -13960.476,E2 -13960.476} C_VEL
LIN {X 0,Y 347.863,Z 891.964,A -85,B 0,C 180,E1 -13964.123,E2 -13964.123} C_VEL
LIN {X 0,Y 347.798,Z 891.972,A -85,B 0,C 180,E1 -13968.241,E2 -13968.241} C_VEL
LIN {X 0,Y 347.767,Z 891.975,A -85,B 0,C 180,E1 -13971.624,E2 -13971.624} C_VEL
LIN {X 0,Y 347.741,Z 891.984,A -85,B 0,C 180,E1 -13975.114,E2 -13975.114} C_VEL
LIN {X 0,Y 347.728,Z 891.981,A -85,B 0,C 180,E1 -13977.701,E2 -13977.701} C_VEL
LIN {X 0,Y 347.74,Z 891.977,A -85,B 0,C 180,E1 -13980.349,E2 -13980.349} C_VEL
LIN {X 0,Y 347.753,Z 891.978,A -85,B 0,C 180,E1 -13984.043,E2 -13984.043} C_VEL
LIN {X 0,Y 347.758,Z 891.978,A -85,B 0,C 180,E1 -13987.322,E2 -13987.322} C_VEL
LIN {X 0,Y 347.7,Z 891.984,A -85,B 0,C 180,E1 -13990.302,E2 -13990.302} C_VEL
LIN {X 0,Y 347.725,Z 891.981,A -85,B 0,C 180,E1 -13993.408,E2 -13993.408} C_VEL
LIN {X 0,Y 347.726,Z 891.98,A -85,B 0,C 180,E1 -13996.687,E2 -13996.687} C_VEL
LIN {X 0,Y 347.704,Z 891.982,A -85,B 0,C 180,E1 -13998.905,E2 -13998.905} C_VEL
LIN {X 0,Y 347.017,Z 892.072,A -85,B 0,C 180,E1 -13999.872,E2 -13999.872} C_VEL
LIN {X 0,Y 344.18,Z 892.421,A -85,B 0,C 180,E1 -14001.445,E2 -14001.445} C_VEL
LIN {X 0,Y 341.796,Z 892.721,A -85,B 0,C 180,E1 -14002.718,E2 -14002.718} C_VEL
LIN {X 0,Y 340.778,Z 892.845,A -85,B 0,C 180,E1 -14003.703,E2 -14003.703} C_VEL
LIN {X 0,Y 340.697,Z 892.854,A -85,B 0,C 180,E1 -14004.036,E2 -14004.036} C_VEL
LIN {X 0,Y 340.69,Z 892.856,A -85,B 0,C 180,E1 -14007.564,E2 -14007.564} C_VEL
LIN {X 0,Y 340.706,Z 892.857,A -85,B 0,C 180,E1 -14010.325,E2 -14010.325} C_VEL
LIN {X 0,Y 340.713,Z 892.857,A -85,B 0,C 180,E1 -14013.011,E2 -14013.011} C_VEL
LIN {X 0,Y 340.703,Z 892.86,A -85,B 0,C 180,E1 -14016.925,E2 -14016.925} C_VEL
LIN {X 0,Y 340.704,Z 892.856,A -85,B 0,C 180,E1 -14020.728,E2 -14020.728} C_VEL
LIN {X 0,Y 340.74,Z 892.856,A -85,B 0,C 180,E1 -14023.216,E2 -14023.216} C_VEL
LIN {X 0,Y 340.838,Z 892.839,A -85,B 0,C 180,E1 -14026.89,E2 -14026.89} C_VEL
LIN {X 0,Y 340.882,Z 892.832,A -85,B 0,C 180,E1 -14030.506,E2 -14030.506} C_VEL
LIN {X 0,Y 341.003,Z 892.817,A -85,B 0,C 180,E1 -14032.896,E2 -14032.896} C_VEL
LIN {X 0,Y 340.802,Z 892.843,A -85,B 0,C 180,E1 -14035.268,E2 -14035.268} C_VEL
LIN {X 0,Y 341.094,Z 892.809,A -85,B 0,C 180,E1 -14037.638,E2 -14037.638} C_VEL
LIN {X 0,Y 341.088,Z 892.806,A -85,B 0,C 180,E1 -14041.18,E2 -14041.18} C_VEL
LIN {X 0,Y 341.093,Z 892.809,A -85,B 0,C 180,E1 -14042.361,E2 -14042.361} C_VEL
LIN {X 0,Y 341.012,Z 892.818,A -85,B 0,C 180,E1 -14045.914,E2 -14045.914} C_VEL
LIN {X 0,Y 340.966,Z 892.828,A -85,B 0,C 180,E1 -14048.356,E2 -14048.356} C_VEL
LIN {X 0,Y 340.844,Z 892.837,A -85,B 0,C 180,E1 -14051.899,E2 -14051.899} C_VEL
LIN {X 0,Y 340.746,Z 892.849,A -85,B 0,C 180,E1 -14055.552,E2 -14055.552} C_VEL
LIN {X 0,Y 340.757,Z 892.85,A -85,B 0,C 180,E1 -14058.424,E2 -14058.424} C_VEL
LIN {X 0,Y 340.719,Z 892.852,A -85,B 0,C 180,E1 -14061.841,E2 -14061.841} C_VEL
LIN {X 0,Y 340.67,Z 892.86,A -85,B 0,C 180,E1 -14065.672,E2 -14065.672} C_VEL
LIN {X 0,Y 340.675,Z 892.857,A -85,B 0,C 180,E1 -14068.325,E2 -14068.325} C_VEL
LIN {X 0,Y 340.692,Z 892.859,A -85,B 0,C 180,E1 -14071.045,E2 -14071.045} C_VEL
LIN {X 0,Y 340.715,Z 892.856,A -85,B 0,C 180,E1 -14075.279,E2 -14075.279} C_VEL
LIN {X 0,Y 340.692,Z 892.856,A -85,B 0,C 180,E1 -14078.382,E2 -14078.382} C_VEL
LIN {X 0,Y 340.69,Z 892.86,A -85,B 0,C 180,E1 -14082.043,E2 -14082.043} C_VEL
LIN {X 0,Y 340.649,Z 892.866,A -85,B 0,C 180,E1 -14086.227,E2 -14086.227} C_VEL
LIN {X 0,Y 340.667,Z 892.86,A -85,B 0,C 180,E1 -14088.687,E2 -14088.687} C_VEL
LIN {X 0,Y 340.717,Z 892.854,A -85,B 0,C 180,E1 -14091.77,E2 -14091.77} C_VEL
LIN {X 0,Y 340.721,Z 892.852,A -85,B 0,C 180,E1 -14095.595,E2 -14095.595} C_VEL
LIN {X 0,Y 340.691,Z 892.859,A -85,B 0,C 180,E1 -14098.954,E2 -14098.954} C_VEL
LIN {X 0,Y 340.758,Z 893.041,A -85,B 0,C 180,E1 -14102.759,E2 -14102.759} C_VEL
LIN {X 0,Y 342.833,Z 904.245,A -85,B 0,C 180,E1 -14106.117,E2 -14106.117} C_VEL
LIN {X 0,Y 342.857,Z 908.32,A -85,B 0,C 180,E1 -14107.282,E2 -14107.282} C_VEL
LIN {X 0,Y 341.607,Z 922.156,A -85,B 0,C 180,E1 -14111.15,E2 -14111.15} C_VEL
LIN {X 0,Y 341.149,Z 927.574,A -85,B 0,C 180,E1 -14112.619,E2 -14112.619} C_VEL
LIN {X 0,Y 344.285,Z 957.418,A -85,B 0,C 180,E1 -14113.57,E2 -14113.57} C_VEL
LIN {X 0,Y 343.306,Z 1006.139,A -85,B 0,C 180,E1 -14114.946,E2 -14114.946} C_VEL
LIN {X 0,Y 342.645,Z 1018.525,A -85,B 0,C 180,E1 -14115.523,E2 -14115.523} C_VEL
LIN {X 0,Y 342.298,Z 1028.24,A -85,B 0,C 180,E1 -14116.191,E2 -14116.191} C_VEL
LIN {X 0,Y 341.735,Z 1036.667,A -85,B 0,C 180,E1 -14116.925,E2 -14116.925} C_VEL
LIN {X 0,Y 341.255,Z 1044.892,A -85,B 0,C 180,E1 -14117.813,E2 -14117.813} C_VEL
LIN {X 0,Y 340.784,Z 1051.709,A -85,B 0,C 180,E1 -14118.701,E2 -14118.701} C_VEL
LIN {X 0,Y 340.235,Z 1059.26,A -85,B 0,C 180,E1 -14119.887,E2 -14119.887} C_VEL
LIN {X 0,Y 339.788,Z 1066.944,A -85,B 0,C 180,E1 -14121.375,E2 -14121.375} C_VEL
LIN {X 0,Y 339.534,Z 1072.92,A -85,B 0,C 180,E1 -14122.866,E2 -14122.866} C_VEL
LIN {X 0,Y 339.276,Z 1076.803,A -85,B 0,C 180,E1 -14124.055,E2 -14124.055} C_VEL
LIN {X 0,Y 339.257,Z 1079.958,A -85,B 0,C 180,E1 -14125.247,E2 -14125.247} C_VEL
LIN {X 0,Y 339.138,Z 1082.392,A -85,B 0,C 180,E1 -14126.435,E2 -14126.435} C_VEL
LIN {X 0,Y 339.088,Z 1084.215,A -85,B 0,C 180,E1 -14127.624,E2 -14127.624} C_VEL
LIN {X 0,Y 339.182,Z 1085.487,A -85,B 0,C 180,E1 -14128.812,E2 -14128.812} C_VEL
LIN {X 0,Y 339.203,Z 1086.219,A -85,B 0,C 180,E1 -14130,E2 -14130} C_VEL
LIN {X 0,Y 339.089,Z 1086.413,A -85,B 0,C 180,E1 -14131.187,E2 -14131.187} C_VEL
LIN {X 0,Y 339.042,Z 1085.991,A -85,B 0,C 180,E1 -14132.376,E2 -14132.376} C_VEL
LIN {X 0,Y 339.123,Z 1084.993,A -85,B 0,C 180,E1 -14133.564,E2 -14133.564} C_VEL
LIN {X 0,Y 339.196,Z 1082.567,A -85,B 0,C 180,E1 -14135.35,E2 -14135.35} C_VEL
LIN {X 0,Y 339.497,Z 1078.762,A -85,B 0,C 180,E1 -14137.135,E2 -14137.135} C_VEL
LIN {X 0,Y 339.881,Z 1074.456,A -85,B 0,C 180,E1 -14138.622,E2 -14138.622} C_VEL
LIN {X 0,Y 340.5,Z 1068.983,A -85,B 0,C 180,E1 -14140.104,E2 -14140.104} C_VEL
LIN {X 0,Y 341.313,Z 1062.155,A -85,B 0,C 180,E1 -14141.581,E2 -14141.581} C_VEL
LIN {X 0,Y 342.237,Z 1053.756,A -85,B 0,C 180,E1 -14143.055,E2 -14143.055} C_VEL
LIN {X 0,Y 343.369,Z 1043.994,A -85,B 0,C 180,E1 -14144.369,E2 -14144.369} C_VEL
LIN {X 0,Y 344.337,Z 1034.536,A -85,B 0,C 180,E1 -14145.387,E2 -14145.387} C_VEL
LIN {X 0,Y 345.503,Z 1023.318,A -85,B 0,C 180,E1 -14146.318,E2 -14146.318} C_VEL
LIN {X 0,Y 346.507,Z 1011.846,A -85,B 0,C 180,E1 -14146.989,E2 -14146.989} C_VEL
LIN {X 0,Y 347.107,Z 1001.71,A -85,B 0,C 180,E1 -14147.414,E2 -14147.414} C_VEL
LIN {X 0,Y 348.788,Z 957.88,A -85,B 0,C 180,E1 -14148.782,E2 -14148.782} C_VEL
LIN {X 0,Y 347.632,Z 945.956,A -85,B 0,C 180,E1 -14149.311,E2 -14149.311} C_VEL
LIN {X 0,Y 345.14,Z 932.837,A -85,B 0,C 180,E1 -14150.038,E2 -14150.038} C_VEL
LIN {X 0,Y 343.141,Z 924.246,A -85,B 0,C 180,E1 -14150.611,E2 -14150.611} C_VEL
LIN {X 0,Y 344.561,Z 914.688,A -85,B 0,C 180,E1 -14153.59,E2 -14153.59} C_VEL
LIN {X 0,Y 344.4,Z 909.574,A -85,B 0,C 180,E1 -14155.375,E2 -14155.375} C_VEL
LIN {X 0,Y 342.987,Z 902.401,A -85,B 0,C 180,E1 -14158.226,E2 -14158.226} C_VEL
LIN {X 0,Y 341.278,Z 895.036,A -85,B 0,C 180,E1 -14161.615,E2 -14161.615} C_VEL
LIN {X 0,Y 340.697,Z 892.862,A -85,B 0,C 180,E1 -14162.785,E2 -14162.785} C_VEL
LIN {X 0,Y 340.704,Z 892.858,A -85,B 0,C 180,E1 -14166.44,E2 -14166.44} C_VEL
LIN {X 0,Y 340.652,Z 892.866,A -85,B 0,C 180,E1 -14169.759,E2 -14169.759} C_VEL
LIN {X 0,Y 340.669,Z 892.863,A -85,B 0,C 180,E1 -14172.905,E2 -14172.905} C_VEL
LIN {X 0,Y 340.669,Z 892.86,A -85,B 0,C 180,E1 -14177.095,E2 -14177.095} C_VEL
LIN {X 0,Y 340.652,Z 892.864,A -85,B 0,C 180,E1 -14180.241,E2 -14180.241} C_VEL
LIN {X 0,Y 340.704,Z 892.857,A -85,B 0,C 180,E1 -14183.561,E2 -14183.561} C_VEL
LIN {X 0,Y 340.69,Z 892.862,A -85,B 0,C 180,E1 -14186.154,E2 -14186.154} C_VEL
LIN {X 0,Y 340.717,Z 892.859,A -85,B 0,C 180,E1 -14190.036,E2 -14190.036} C_VEL
LIN {X 0,Y 340.715,Z 892.892,A -85,B 0,C 180,E1 -14193.344,E2 -14193.344} C_VEL
LIN {X 0,Y 341.955,Z 898.266,A -85,B 0,C 180,E1 -14196.374,E2 -14196.374} C_VEL
LIN {X 0,Y 343.17,Z 904.612,A -85,B 0,C 180,E1 -14199.509,E2 -14199.509} C_VEL
LIN {X 0,Y 346.979,Z 913.677,A -85,B 0,C 180,E1 -14200.266,E2 -14200.266} C_VEL
LIN {X 0,Y 349.564,Z 923.6,A -85,B 0,C 180,E1 -14200.898,E2 -14200.898} C_VEL
LIN {X 0,Y 349.835,Z 926.478,A -85,B 0,C 180,E1 -14201.027,E2 -14201.027} C_VEL
LIN {X 0,Y 347.318,Z 982.172,A -85,B 0,C 180,E1 -14202.787,E2 -14202.787} C_VEL
LIN {X 0,Y 346.635,Z 994.321,A -85,B 0,C 180,E1 -14203.435,E2 -14203.435} C_VEL
LIN {X 0,Y 345.892,Z 1003.333,A -85,B 0,C 180,E1 -14204.08,E2 -14204.08} C_VEL
LIN {X 0,Y 345.056,Z 1012.775,A -85,B 0,C 180,E1 -14204.949,E2 -14204.949} C_VEL
LIN {X 0,Y 344.065,Z 1022.731,A -85,B 0,C 180,E1 -14206.113,E2 -14206.113} C_VEL
LIN {X 0,Y 343.162,Z 1030.537,A -85,B 0,C 180,E1 -14207.282,E2 -14207.282} C_VEL
LIN {X 0,Y 342.358,Z 1036.978,A -85,B 0,C 180,E1 -14208.455,E2 -14208.455} C_VEL
LIN {X 0,Y 341.556,Z 1042.358,A -85,B 0,C 180,E1 -14209.628,E2 -14209.628} C_VEL
LIN {X 0,Y 340.91,Z 1047.802,A -85,B 0,C 180,E1 -14211.106,E2 -14211.106} C_VEL
LIN {X 0,Y 340.554,Z 1050.908,A -85,B 0,C 180,E1 -14212.127,E2 -14212.127} C_VEL
LIN {X 0,Y 340.053,Z 1054.209,A -85,B 0,C 180,E1 -14213.474,E2 -14213.474} C_VEL
LIN {X 0,Y 339.541,Z 1057.29,A -85,B 0,C 180,E1 -14215.251,E2 -14215.251} C_VEL
LIN {X 0,Y 339.457,Z 1058.654,A -85,B 0,C 180,E1 -14216.44,E2 -14216.44} C_VEL
LIN {X 0,Y 339.348,Z 1059.505,A -85,B 0,C 180,E1 -14217.627,E2 -14217.627} C_VEL
LIN {X 0,Y 339.217,Z 1059.767,A -85,B 0,C 180,E1 -14218.813,E2 -14218.813} C_VEL
LIN {X 0,Y 339.14,Z 1059.439,A -85,B 0,C 180,E1 -14220.001,E2 -14220.001} C_VEL
LIN {X 0,Y 339.109,Z 1058.599,A -85,B 0,C 180,E1 -14221.188,E2 -14221.188} C_VEL
LIN {X 0,Y 339.137,Z 1057.234,A -85,B 0,C 180,E1 -14222.376,E2 -14222.376} C_VEL
LIN {X 0,Y 339.311,Z 1054.069,A -85,B 0,C 180,E1 -14224.158,E2 -14224.158} C_VEL
LIN {X 0,Y 339.421,Z 1051.188,A -85,B 0,C 180,E1 -14225.347,E2 -14225.347} C_VEL
LIN {X 0,Y 339.696,Z 1046.13,A -85,B 0,C 180,E1 -14226.974,E2 -14226.974} C_VEL
LIN {X 0,Y 340.068,Z 1039.548,A -85,B 0,C 180,E1 -14228.618,E2 -14228.618} C_VEL
LIN {X 0,Y 340.611,Z 1031.8,A -85,B 0,C 180,E1 -14230.102,E2 -14230.102} C_VEL
LIN {X 0,Y 341.078,Z 1024.161,A -85,B 0,C 180,E1 -14231.289,E2 -14231.289} C_VEL
LIN {X 0,Y 341.611,Z 1016.027,A -85,B 0,C 180,E1 -14232.325,E2 -14232.325} C_VEL
LIN {X 0,Y 342.265,Z 1005.944,A -85,B 0,C 180,E1 -14233.357,E2 -14233.357} C_VEL
LIN {X 0,Y 342.747,Z 995.323,A -85,B 0,C 180,E1 -14234.169,E2 -14234.169} C_VEL
LIN {X 0,Y 343.002,Z 985.659,A -85,B 0,C 180,E1 -14234.727,E2 -14234.727} C_VEL
LIN {X 0,Y 343.395,Z 975.743,A -85,B 0,C 180,E1 -14235.127,E2 -14235.127} C_VEL
LIN {X 0,Y 344.52,Z 921.716,A -85,B 0,C 180,E1 -14236.626,E2 -14236.626} C_VEL
LIN {X 0,Y 341.265,Z 900.678,A -85,B 0,C 180,E1 -14237.331,E2 -14237.331} C_VEL
LIN {X 0,Y 341.307,Z 896.659,A -85,B 0,C 180,E1 -14238.701,E2 -14238.701} C_VEL
LIN {X 0,Y 340.854,Z 892.837,A -85,B 0,C 180,E1 -14240.047,E2 -14240.047} C_VEL
LIN {X 0,Y 340.716,Z 892.853,A -85,B 0,C 180,E1 -14244.365,E2 -14244.365} C_VEL
LIN {X 0,Y 340.687,Z 892.86,A -85,B 0,C 180,E1 -14247.496,E2 -14247.496} C_VEL
LIN {X 0,Y 340.694,Z 892.858,A -85,B 0,C 180,E1 -14251.046,E2 -14251.046} C_VEL
LIN {X 0,Y 340.717,Z 892.856,A -85,B 0,C 180,E1 -14255.28,E2 -14255.28} C_VEL
LIN {X 0,Y 340.695,Z 892.856,A -85,B 0,C 180,E1 -14258.383,E2 -14258.383} C_VEL
LIN {X 0,Y 340.692,Z 892.86,A -85,B 0,C 180,E1 -14262.044,E2 -14262.044} C_VEL
LIN {X 0,Y 340.651,Z 892.865,A -85,B 0,C 180,E1 -14266.228,E2 -14266.228} C_VEL
LIN {X 0,Y 340.67,Z 892.86,A -85,B 0,C 180,E1 -14268.688,E2 -14268.688} C_VEL
LIN {X 0,Y 340.72,Z 892.854,A -85,B 0,C 180,E1 -14271.771,E2 -14271.771} C_VEL
LIN {X 0,Y 340.725,Z 892.851,A -85,B 0,C 180,E1 -14275.596,E2 -14275.596} C_VEL
LIN {X 0,Y 340.695,Z 892.858,A -85,B 0,C 180,E1 -14278.955,E2 -14278.955} C_VEL
LIN {X 0,Y 340.714,Z 892.857,A -85,B 0,C 180,E1 -14283.012,E2 -14283.012} C_VEL
LIN {X 0,Y 340.742,Z 892.85,A -85,B 0,C 180,E1 -14285.637,E2 -14285.637} C_VEL
LIN {X 0,Y 340.713,Z 892.856,A -85,B 0,C 180,E1 -14289.472,E2 -14289.472} C_VEL
LIN {X 0,Y 340.762,Z 892.853,A -85,B 0,C 180,E1 -14293.218,E2 -14293.218} C_VEL
LIN {X 0,Y 340.857,Z 892.838,A -85,B 0,C 180,E1 -14295.717,E2 -14295.717} C_VEL
LIN {X 0,Y 340.846,Z 892.841,A -85,B 0,C 180,E1 -14299.306,E2 -14299.306} C_VEL
LIN {X 0,Y 341.004,Z 892.817,A -85,B 0,C 180,E1 -14302.897,E2 -14302.897} C_VEL
LIN {X 0,Y 340.804,Z 892.843,A -85,B 0,C 180,E1 -14305.269,E2 -14305.269} C_VEL
LIN {X 0,Y 341.096,Z 892.809,A -85,B 0,C 180,E1 -14307.638,E2 -14307.638} C_VEL
LIN {X 0,Y 341.091,Z 892.806,A -85,B 0,C 180,E1 -14311.181,E2 -14311.181} C_VEL
LIN {X 0,Y 341.095,Z 892.809,A -85,B 0,C 180,E1 -14312.362,E2 -14312.362} C_VEL
LIN {X 0,Y 341.015,Z 892.818,A -85,B 0,C 180,E1 -14315.915,E2 -14315.915} C_VEL
LIN {X 0,Y 340.969,Z 892.827,A -85,B 0,C 180,E1 -14318.356,E2 -14318.356} C_VEL
LIN {X 0,Y 340.847,Z 892.837,A -85,B 0,C 180,E1 -14321.9,E2 -14321.9} C_VEL
LIN {X 0,Y 340.749,Z 892.848,A -85,B 0,C 180,E1 -14325.553,E2 -14325.553} C_VEL
LIN {X 0,Y 340.76,Z 892.85,A -85,B 0,C 180,E1 -14328.425,E2 -14328.425} C_VEL
LIN {X 0,Y 340.723,Z 892.852,A -85,B 0,C 180,E1 -14331.842,E2 -14331.842} C_VEL
LIN {X 0,Y 340.674,Z 892.859,A -85,B 0,C 180,E1 -14335.673,E2 -14335.673} C_VEL
LIN {X 0,Y 340.679,Z 892.857,A -85,B 0,C 180,E1 -14338.326,E2 -14338.326} C_VEL
LIN {X 0,Y 340.696,Z 892.858,A -85,B 0,C 180,E1 -14341.045,E2 -14341.045} C_VEL
LIN {X 0,Y 340.719,Z 892.856,A -85,B 0,C 180,E1 -14345.279,E2 -14345.279} C_VEL
LIN {X 0,Y 340.697,Z 892.856,A -85,B 0,C 180,E1 -14348.382,E2 -14348.382} C_VEL
LIN {X 0,Y 340.694,Z 892.86,A -85,B 0,C 180,E1 -14352.043,E2 -14352.043} C_VEL
LIN {X 0,Y 340.653,Z 892.865,A -85,B 0,C 180,E1 -14356.227,E2 -14356.227} C_VEL
LIN {X 0,Y 340.659,Z 892.86,A -85,B 0,C 180,E1 -14358.895,E2 -14358.895} C_VEL
LIN {X 0,Y 340.721,Z 892.853,A -85,B 0,C 180,E1 -14361.77,E2 -14361.77} C_VEL
LIN {X 0,Y 340.697,Z 892.854,A -85,B 0,C 180,E1 -14364.036,E2 -14364.036} C_VEL
LIN {X 0,Y 340.023,Z 892.942,A -85,B 0,C 180,E1 -14365.024,E2 -14365.024} C_VEL
LIN {X 0,Y 337.135,Z 893.304,A -85,B 0,C 180,E1 -14366.629,E2 -14366.629} C_VEL
LIN {X 0,Y 334.709,Z 893.602,A -85,B 0,C 180,E1 -14367.93,E2 -14367.93} C_VEL
LIN {X 0,Y 333.699,Z 893.73,A -85,B 0,C 180,E1 -14368.937,E2 -14368.937} C_VEL
LIN {X 0,Y 333.634,Z 893.733,A -85,B 0,C 180,E1 -14369.278,E2 -14369.278} C_VEL
LIN {X 0,Y 333.663,Z 893.734,A -85,B 0,C 180,E1 -14372.393,E2 -14372.393} C_VEL
LIN {X 0,Y 333.666,Z 893.735,A -85,B 0,C 180,E1 -14375.085,E2 -14375.085} C_VEL
LIN {X 0,Y 333.654,Z 893.738,A -85,B 0,C 180,E1 -14379.017,E2 -14379.017} C_VEL
LIN {X 0,Y 333.714,Z 893.727,A -85,B 0,C 180,E1 -14381.584,E2 -14381.584} C_VEL
LIN {X 0,Y 333.764,Z 893.722,A -85,B 0,C 180,E1 -14385.608,E2 -14385.608} C_VEL
LIN {X 0,Y 333.815,Z 893.714,A -85,B 0,C 180,E1 -14389.077,E2 -14389.077} C_VEL
LIN {X 0,Y 333.958,Z 893.694,A -85,B 0,C 180,E1 -14392.745,E2 -14392.745} C_VEL
LIN {X 0,Y 333.77,Z 893.719,A -85,B 0,C 180,E1 -14395.168,E2 -14395.168} C_VEL
LIN {X 0,Y 334.037,Z 893.688,A -85,B 0,C 180,E1 -14397.588,E2 -14397.588} C_VEL
LIN {X 0,Y 334.058,Z 893.682,A -85,B 0,C 180,E1 -14401.205,E2 -14401.205} C_VEL
LIN {X 0,Y 333.777,Z 893.718,A -85,B 0,C 180,E1 -14403.621,E2 -14403.621} C_VEL
LIN {X 0,Y 333.987,Z 893.695,A -85,B 0,C 180,E1 -14406.039,E2 -14406.039} C_VEL
LIN {X 0,Y 333.915,Z 893.705,A -85,B 0,C 180,E1 -14408.472,E2 -14408.472} C_VEL
LIN {X 0,Y 333.785,Z 893.718,A -85,B 0,C 180,E1 -14412.154,E2 -14412.154} C_VEL
LIN {X 0,Y 333.737,Z 893.728,A -85,B 0,C 180,E1 -14414.637,E2 -14414.637} C_VEL
LIN {X 0,Y 333.696,Z 893.731,A -85,B 0,C 180,E1 -14418.602,E2 -14418.602} C_VEL
LIN {X 0,Y 333.65,Z 893.733,A -85,B 0,C 180,E1 -14422.281,E2 -14422.281} C_VEL
LIN {X 0,Y 333.658,Z 893.738,A -85,B 0,C 180,E1 -14425.077,E2 -14425.077} C_VEL
LIN {X 0,Y 333.649,Z 893.736,A -85,B 0,C 180,E1 -14428.977,E2 -14428.977} C_VEL
LIN {X 0,Y 333.644,Z 893.734,A -85,B 0,C 180,E1 -14432.586,E2 -14432.586} C_VEL
LIN {X 0,Y 333.673,Z 893.731,A -85,B 0,C 180,E1 -14436.139,E2 -14436.139} C_VEL
LIN {X 0,Y 333.601,Z 893.74,A -85,B 0,C 180,E1 -14439.198,E2 -14439.198} C_VEL
LIN {X 0,Y 333.626,Z 893.737,A -85,B 0,C 180,E1 -14442.498,E2 -14442.498} C_VEL
LIN {X 0,Y 333.593,Z 893.745,A -85,B 0,C 180,E1 -14445.954,E2 -14445.954} C_VEL
LIN {X 0,Y 333.601,Z 893.739,A -85,B 0,C 180,E1 -14449.324,E2 -14449.324} C_VEL
LIN {X 0,Y 333.66,Z 893.732,A -85,B 0,C 180,E1 -14453.168,E2 -14453.168} C_VEL
LIN {X 0,Y 333.672,Z 893.73,A -85,B 0,C 180,E1 -14455.341,E2 -14455.341} C_VEL
LIN {X 0,Y 333.628,Z 893.738,A -85,B 0,C 180,E1 -14458.221,E2 -14458.221} C_VEL
LIN {X 0,Y 333.652,Z 893.736,A -85,B 0,C 180,E1 -14461.022,E2 -14461.022} C_VEL
LIN {X 0,Y 333.709,Z 893.861,A -85,B 0,C 180,E1 -14462.61,E2 -14462.61} C_VEL
LIN {X 0,Y 335.702,Z 904.606,A -85,B 0,C 180,E1 -14465.906,E2 -14465.906} C_VEL
LIN {X 0,Y 335.875,Z 908.415,A -85,B 0,C 180,E1 -14467.024,E2 -14467.024} C_VEL
LIN {X 0,Y 334.591,Z 922.134,A -85,B 0,C 180,E1 -14470.945,E2 -14470.945} C_VEL
LIN {X 0,Y 334.106,Z 927.13,A -85,B 0,C 180,E1 -14472.359,E2 -14472.359} C_VEL
LIN {X 0,Y 337.278,Z 958.587,A -85,B 0,C 180,E1 -14473.418,E2 -14473.418} C_VEL
LIN {X 0,Y 336.286,Z 1005.433,A -85,B 0,C 180,E1 -14474.779,E2 -14474.779} C_VEL
LIN {X 0,Y 335.683,Z 1016.734,A -85,B 0,C 180,E1 -14475.294,E2 -14475.294} C_VEL
LIN {X 0,Y 335.265,Z 1027.744,A -85,B 0,C 180,E1 -14476.05,E2 -14476.05} C_VEL
LIN {X 0,Y 334.694,Z 1036.206,A -85,B 0,C 180,E1 -14476.799,E2 -14476.799} C_VEL
LIN {X 0,Y 334.2,Z 1044.46,A -85,B 0,C 180,E1 -14477.706,E2 -14477.706} C_VEL
LIN {X 0,Y 333.706,Z 1051.301,A -85,B 0,C 180,E1 -14478.612,E2 -14478.612} C_VEL
LIN {X 0,Y 333.23,Z 1058.009,A -85,B 0,C 180,E1 -14479.673,E2 -14479.673} C_VEL
LIN {X 0,Y 332.838,Z 1064.402,A -85,B 0,C 180,E1 -14480.888,E2 -14480.888} C_VEL
LIN {X 0,Y 332.494,Z 1070.917,A -85,B 0,C 180,E1 -14482.408,E2 -14482.408} C_VEL
LIN {X 0,Y 332.18,Z 1077.119,A -85,B 0,C 180,E1 -14484.323,E2 -14484.323} C_VEL
LIN {X 0,Y 332.154,Z 1080.592,A -85,B 0,C 180,E1 -14485.753,E2 -14485.753} C_VEL
LIN {X 0,Y 332.001,Z 1083.696,A -85,B 0,C 180,E1 -14487.573,E2 -14487.573} C_VEL
LIN {X 0,Y 332.087,Z 1085.052,A -85,B 0,C 180,E1 -14488.787,E2 -14488.787} C_VEL
LIN {X 0,Y 332.11,Z 1085.867,A -85,B 0,C 180,E1 -14490,E2 -14490} C_VEL
LIN {X 0,Y 331.992,Z 1086.107,A -85,B 0,C 180,E1 -14491.213,E2 -14491.213} C_VEL
LIN {X 0,Y 331.958,Z 1085.724,A -85,B 0,C 180,E1 -14492.427,E2 -14492.427} C_VEL
LIN {X 0,Y 332.051,Z 1084.817,A -85,B 0,C 180,E1 -14493.64,E2 -14493.64} C_VEL
LIN {X 0,Y 332.107,Z 1083.383,A -85,B 0,C 180,E1 -14494.856,E2 -14494.856} C_VEL
LIN {X 0,Y 332.315,Z 1080.135,A -85,B 0,C 180,E1 -14496.679,E2 -14496.679} C_VEL
LIN {X 0,Y 332.779,Z 1075.55,A -85,B 0,C 180,E1 -14498.501,E2 -14498.501} C_VEL
LIN {X 0,Y 333.536,Z 1069.294,A -85,B 0,C 180,E1 -14500.317,E2 -14500.317} C_VEL
LIN {X 0,Y 334.189,Z 1064.121,A -85,B 0,C 180,E1 -14501.524,E2 -14501.524} C_VEL
LIN {X 0,Y 334.984,Z 1057.92,A -85,B 0,C 180,E1 -14502.726,E2 -14502.726} C_VEL
LIN {X 0,Y 335.912,Z 1050.431,A -85,B 0,C 180,E1 -14503.922,E2 -14503.922} C_VEL
LIN {X 0,Y 336.859,Z 1042.507,A -85,B 0,C 180,E1 -14504.962,E2 -14504.962} C_VEL
LIN {X 0,Y 337.943,Z 1032.867,A -85,B 0,C 180,E1 -14505.995,E2 -14505.995} C_VEL
LIN {X 0,Y 339.232,Z 1021.14,A -85,B 0,C 180,E1 -14506.938,E2 -14506.938} C_VEL
LIN {X 0,Y 340.159,Z 1010.758,A -85,B 0,C 180,E1 -14507.549,E2 -14507.549} C_VEL
LIN {X 0,Y 340.858,Z 999.636,A -85,B 0,C 180,E1 -14508.016,E2 -14508.016} C_VEL
LIN {X 0,Y 342.525,Z 958.59,A -85,B 0,C 180,E1 -14509.328,E2 -14509.328} C_VEL
LIN {X 0,Y 341.43,Z 947.014,A -85,B 0,C 180,E1 -14509.876,E2 -14509.876} C_VEL
LIN {X 0,Y 338.987,Z 934.044,A -85,B 0,C 180,E1 -14510.637,E2 -14510.637} C_VEL
LIN {X 0,Y 336.528,Z 923.915,A -85,B 0,C 180,E1 -14511.336,E2 -14511.336} C_VEL
LIN {X 0,Y 337.806,Z 915.628,A -85,B 0,C 180,E1 -14514.019,E2 -14514.019} C_VEL
LIN {X 0,Y 337.704,Z 912.204,A -85,B 0,C 180,E1 -14515.254,E2 -14515.254} C_VEL
LIN {X 0,Y 336.47,Z 905.526,A -85,B 0,C 180,E1 -14517.956,E2 -14517.956} C_VEL
LIN {X 0,Y 335.145,Z 899.564,A -85,B 0,C 180,E1 -14520.71,E2 -14520.71} C_VEL
LIN {X 0,Y 333.661,Z 893.738,A -85,B 0,C 180,E1 -14523.93,E2 -14523.93} C_VEL
LIN {X 0,Y 333.639,Z 893.738,A -85,B 0,C 180,E1 -14527.653,E2 -14527.653} C_VEL
LIN {X 0,Y 333.6,Z 893.741,A -85,B 0,C 180,E1 -14530.774,E2 -14530.774} C_VEL
LIN {X 0,Y 333.587,Z 893.745,A -85,B 0,C 180,E1 -14534.25,E2 -14534.25} C_VEL
LIN {X 0,Y 333.633,Z 893.739,A -85,B 0,C 180,E1 -14537.618,E2 -14537.618} C_VEL
LIN {X 0,Y 333.613,Z 893.742,A -85,B 0,C 180,E1 -14541.21,E2 -14541.21} C_VEL
LIN {X 0,Y 333.671,Z 893.733,A -85,B 0,C 180,E1 -14543.861,E2 -14543.861} C_VEL
LIN {X 0,Y 333.642,Z 893.74,A -85,B 0,C 180,E1 -14547.414,E2 -14547.414} C_VEL
LIN {X 0,Y 333.626,Z 893.741,A -85,B 0,C 180,E1 -14551.02,E2 -14551.02} C_VEL
LIN {X 0,Y 333.67,Z 893.904,A -85,B 0,C 180,E1 -14552.34,E2 -14552.34} C_VEL
LIN {X 0,Y 335.079,Z 899.693,A -85,B 0,C 180,E1 -14555.859,E2 -14555.859} C_VEL
LIN {X 0,Y 336.133,Z 905.11,A -85,B 0,C 180,E1 -14558.699,E2 -14558.699} C_VEL
LIN {X 0,Y 340.843,Z 915.448,A -85,B 0,C 180,E1 -14559.68,E2 -14559.68} C_VEL
LIN {X 0,Y 343.365,Z 924.646,A -85,B 0,C 180,E1 -14560.31,E2 -14560.31} C_VEL
LIN {X 0,Y 343.706,Z 927.287,A -85,B 0,C 180,E1 -14560.447,E2 -14560.447} C_VEL
LIN {X 0,Y 340.98,Z 982.637,A -85,B 0,C 180,E1 -14562.263,E2 -14562.263} C_VEL
LIN {X 0,Y 340.292,Z 994.191,A -85,B 0,C 180,E1 -14562.885,E2 -14562.885} C_VEL
LIN {X 0,Y 339.426,Z 1004.08,A -85,B 0,C 180,E1 -14563.614,E2 -14563.614} C_VEL
LIN {X 0,Y 338.51,Z 1013.367,A -85,B 0,C 180,E1 -14564.497,E2 -14564.497} C_VEL
LIN {X 0,Y 337.457,Z 1023.187,A -85,B 0,C 180,E1 -14565.682,E2 -14565.682} C_VEL
LIN {X 0,Y 336.353,Z 1031.815,A -85,B 0,C 180,E1 -14567.02,E2 -14567.02} C_VEL
LIN {X 0,Y 335.494,Z 1038.12,A -85,B 0,C 180,E1 -14568.215,E2 -14568.215} C_VEL
LIN {X 0,Y 334.665,Z 1043.373,A -85,B 0,C 180,E1 -14569.412,E2 -14569.412} C_VEL
LIN {X 0,Y 333.965,Z 1048.689,A -85,B 0,C 180,E1 -14570.92,E2 -14570.92} C_VEL
LIN {X 0,Y 333.566,Z 1051.754,A -85,B 0,C 180,E1 -14571.995,E2 -14571.995} C_VEL
LIN {X 0,Y 333.042,Z 1054.852,A -85,B 0,C 180,E1 -14573.336,E2 -14573.336} C_VEL
LIN {X 0,Y 332.487,Z 1057.835,A -85,B 0,C 180,E1 -14575.15,E2 -14575.15} C_VEL
LIN {X 0,Y 332.379,Z 1059.109,A -85,B 0,C 180,E1 -14576.364,E2 -14576.364} C_VEL
LIN {X 0,Y 332.261,Z 1059.871,A -85,B 0,C 180,E1 -14577.576,E2 -14577.576} C_VEL
LIN {X 0,Y 332.127,Z 1060.097,A -85,B 0,C 180,E1 -14578.788,E2 -14578.788} C_VEL
LIN {X 0,Y 332.045,Z 1059.699,A -85,B 0,C 180,E1 -14580.001,E2 -14580.001} C_VEL
LIN {X 0,Y 332.012,Z 1058.761,A -85,B 0,C 180,E1 -14581.213,E2 -14581.213} C_VEL
LIN {X 0,Y 332.083,Z 1056.398,A -85,B 0,C 180,E1 -14583.033,E2 -14583.033} C_VEL
LIN {X 0,Y 332.293,Z 1052.666,A -85,B 0,C 180,E1 -14584.854,E2 -14584.854} C_VEL
LIN {X 0,Y 332.489,Z 1047.776,A -85,B 0,C 180,E1 -14586.554,E2 -14586.554} C_VEL
LIN {X 0,Y 332.826,Z 1042.928,A -85,B 0,C 180,E1 -14587.89,E2 -14587.89} C_VEL
LIN {X 0,Y 333.116,Z 1037.576,A -85,B 0,C 180,E1 -14589.105,E2 -14589.105} C_VEL
LIN {X 0,Y 333.569,Z 1031.118,A -85,B 0,C 180,E1 -14590.317,E2 -14590.317} C_VEL
LIN {X 0,Y 334.109,Z 1023.29,A -85,B 0,C 180,E1 -14591.528,E2 -14591.528} C_VEL
LIN {X 0,Y 334.762,Z 1013.611,A -85,B 0,C 180,E1 -14592.735,E2 -14592.735} C_VEL
LIN {X 0,Y 335.303,Z 1004.232,A -85,B 0,C 180,E1 -14593.639,E2 -14593.639} C_VEL
LIN {X 0,Y 335.789,Z 994.215,A -85,B 0,C 180,E1 -14594.392,E2 -14594.392} C_VEL
LIN {X 0,Y 336.019,Z 984.133,A -85,B 0,C 180,E1 -14594.962,E2 -14594.962} C_VEL
LIN {X 0,Y 336.494,Z 970.91,A -85,B 0,C 180,E1 -14595.445,E2 -14595.445} C_VEL
LIN {X 0,Y 337.515,Z 922.232,A -85,B 0,C 180,E1 -14596.819,E2 -14596.819} C_VEL
LIN {X 0,Y 334.239,Z 900.94,A -85,B 0,C 180,E1 -14597.554,E2 -14597.554} C_VEL
LIN {X 0,Y 334.154,Z 896.25,A -85,B 0,C 180,E1 -14599.195,E2 -14599.195} C_VEL
LIN {X 0,Y 333.793,Z 893.716,A -85,B 0,C 180,E1 -14600.169,E2 -14600.169} C_VEL
LIN {X 0,Y 333.664,Z 893.735,A -85,B 0,C 180,E1 -14604.915,E2 -14604.915} C_VEL
LIN {X 0,Y 333.65,Z 893.736,A -85,B 0,C 180,E1 -14608.979,E2 -14608.979} C_VEL
LIN {X 0,Y 333.645,Z 893.733,A -85,B 0,C 180,E1 -14612.587,E2 -14612.587} C_VEL
LIN {X 0,Y 333.675,Z 893.731,A -85,B 0,C 180,E1 -14616.14,E2 -14616.14} C_VEL
LIN {X 0,Y 333.603,Z 893.74,A -85,B 0,C 180,E1 -14619.199,E2 -14619.199} C_VEL
LIN {X 0,Y 333.628,Z 893.736,A -85,B 0,C 180,E1 -14622.499,E2 -14622.499} C_VEL
LIN {X 0,Y 333.595,Z 893.745,A -85,B 0,C 180,E1 -14625.955,E2 -14625.955} C_VEL
LIN {X 0,Y 333.604,Z 893.739,A -85,B 0,C 180,E1 -14629.325,E2 -14629.325} C_VEL
LIN {X 0,Y 333.664,Z 893.731,A -85,B 0,C 180,E1 -14633.169,E2 -14633.169} C_VEL
LIN {X 0,Y 333.676,Z 893.73,A -85,B 0,C 180,E1 -14635.342,E2 -14635.342} C_VEL
LIN {X 0,Y 333.632,Z 893.738,A -85,B 0,C 180,E1 -14638.222,E2 -14638.222} C_VEL
LIN {X 0,Y 333.653,Z 893.736,A -85,B 0,C 180,E1 -14641.023,E2 -14641.023} C_VEL
LIN {X 0,Y 333.698,Z 893.731,A -85,B 0,C 180,E1 -14645.089,E2 -14645.089} C_VEL
LIN {X 0,Y 333.655,Z 893.738,A -85,B 0,C 180,E1 -14649.018,E2 -14649.018} C_VEL
LIN {X 0,Y 333.702,Z 893.729,A -85,B 0,C 180,E1 -14652.852,E2 -14652.852} C_VEL
LIN {X 0,Y 333.813,Z 893.717,A -85,B 0,C 180,E1 -14655.577,E2 -14655.577} C_VEL
LIN {X 0,Y 333.817,Z 893.714,A -85,B 0,C 180,E1 -14659.078,E2 -14659.078} C_VEL
LIN {X 0,Y 333.96,Z 893.694,A -85,B 0,C 180,E1 -14662.746,E2 -14662.746} C_VEL
LIN {X 0,Y 333.772,Z 893.718,A -85,B 0,C 180,E1 -14665.169,E2 -14665.169} C_VEL
LIN {X 0,Y 334.04,Z 893.687,A -85,B 0,C 180,E1 -14667.589,E2 -14667.589} C_VEL
LIN {X 0,Y 334.061,Z 893.682,A -85,B 0,C 180,E1 -14671.206,E2 -14671.206} C_VEL
LIN {X 0,Y 333.779,Z 893.718,A -85,B 0,C 180,E1 -14673.622,E2 -14673.622} C_VEL
LIN {X 0,Y 333.989,Z 893.695,A -85,B 0,C 180,E1 -14676.04,E2 -14676.04} C_VEL
LIN {X 0,Y 333.918,Z 893.705,A -85,B 0,C 180,E1 -14678.472,E2 -14678.472} C_VEL
LIN {X 0,Y 333.788,Z 893.718,A -85,B 0,C 180,E1 -14682.155,E2 -14682.155} C_VEL
LIN {X 0,Y 333.741,Z 893.728,A -85,B 0,C 180,E1 -14684.638,E2 -14684.638} C_VEL
LIN {X 0,Y 333.699,Z 893.731,A -85,B 0,C 180,E1 -14688.603,E2 -14688.603} C_VEL
LIN {X 0,Y 333.653,Z 893.733,A -85,B 0,C 180,E1 -14692.281,E2 -14692.281} C_VEL
LIN {X 0,Y 333.662,Z 893.737,A -85,B 0,C 180,E1 -14695.078,E2 -14695.078} C_VEL
LIN {X 0,Y 333.653,Z 893.736,A -85,B 0,C 180,E1 -14698.978,E2 -14698.978} C_VEL
LIN {X 0,Y 333.648,Z 893.733,A -85,B 0,C 180,E1 -14702.587,E2 -14702.587} C_VEL
LIN {X 0,Y 333.677,Z 893.731,A -85,B 0,C 180,E1 -14706.139,E2 -14706.139} C_VEL
LIN {X 0,Y 333.605,Z 893.74,A -85,B 0,C 180,E1 -14709.199,E2 -14709.199} C_VEL
LIN {X 0,Y 333.63,Z 893.736,A -85,B 0,C 180,E1 -14712.498,E2 -14712.498} C_VEL
LIN {X 0,Y 333.597,Z 893.745,A -85,B 0,C 180,E1 -14715.954,E2 -14715.954} C_VEL
LIN {X 0,Y 333.605,Z 893.738,A -85,B 0,C 180,E1 -14719.324,E2 -14719.324} C_VEL
LIN {X 0,Y 333.665,Z 893.731,A -85,B 0,C 180,E1 -14723.169,E2 -14723.169} C_VEL
LIN {X 0,Y 333.677,Z 893.729,A -85,B 0,C 180,E1 -14725.341,E2 -14725.341} C_VEL
LIN {X 0,Y 333.634,Z 893.733,A -85,B 0,C 180,E1 -14729.278,E2 -14729.278} C_VEL
LIN {X 0,Y 333.015,Z 893.816,A -85,B 0,C 180,E1 -14730.285,E2 -14730.285} C_VEL
LIN {X 0,Y 330.187,Z 894.164,A -85,B 0,C 180,E1 -14731.924,E2 -14731.924} C_VEL
LIN {X 0,Y 327.752,Z 894.469,A -85,B 0,C 180,E1 -14733.251,E2 -14733.251} C_VEL
LIN {X 0,Y 326.691,Z 894.601,A -85,B 0,C 180,E1 -14734.279,E2 -14734.279} C_VEL
LIN {X 0,Y 326.598,Z 894.615,A -85,B 0,C 180,E1 -14734.627,E2 -14734.627} C_VEL
LIN {X 0,Y 326.611,Z 894.611,A -85,B 0,C 180,E1 -14738.542,E2 -14738.542} C_VEL
LIN {X 0,Y 326.632,Z 894.607,A -85,B 0,C 180,E1 -14742.468,E2 -14742.468} C_VEL
LIN {X 0,Y 326.735,Z 894.594,A -85,B 0,C 180,E1 -14746.313,E2 -14746.313} C_VEL
LIN {X 0,Y 326.783,Z 894.589,A -85,B 0,C 180,E1 -14750.092,E2 -14750.092} C_VEL
LIN {X 0,Y 326.942,Z 894.574,A -85,B 0,C 180,E1 -14753.829,E2 -14753.829} C_VEL
LIN {X 0,Y 326.984,Z 894.566,A -85,B 0,C 180,E1 -14757.536,E2 -14757.536} C_VEL
LIN {X 0,Y 327.028,Z 894.558,A -85,B 0,C 180,E1 -14761.231,E2 -14761.231} C_VEL
LIN {X 0,Y 326.727,Z 894.597,A -85,B 0,C 180,E1 -14763.699,E2 -14763.699} C_VEL
LIN {X 0,Y 326.941,Z 894.574,A -85,B 0,C 180,E1 -14766.17,E2 -14766.17} C_VEL
LIN {X 0,Y 326.782,Z 894.59,A -85,B 0,C 180,E1 -14769.907,E2 -14769.907} C_VEL
LIN {X 0,Y 326.734,Z 894.594,A -85,B 0,C 180,E1 -14773.686,E2 -14773.686} C_VEL
LIN {X 0,Y 326.63,Z 894.607,A -85,B 0,C 180,E1 -14777.531,E2 -14777.531} C_VEL
LIN {X 0,Y 326.609,Z 894.611,A -85,B 0,C 180,E1 -14781.457,E2 -14781.457} C_VEL
LIN {X 0,Y 326.6,Z 894.614,A -85,B 0,C 180,E1 -14785.491,E2 -14785.491} C_VEL
LIN {X 0,Y 326.614,Z 894.612,A -85,B 0,C 180,E1 -14789.663,E2 -14789.663} C_VEL
LIN {X 0,Y 326.617,Z 894.61,A -85,B 0,C 180,E1 -14792.945,E2 -14792.945} C_VEL
LIN {X 0,Y 326.611,Z 894.615,A -85,B 0,C 180,E1 -14795.519,E2 -14795.519} C_VEL
LIN {X 0,Y 326.571,Z 894.616,A -85,B 0,C 180,E1 -14799.218,E2 -14799.218} C_VEL
LIN {X 0,Y 326.571,Z 894.614,A -85,B 0,C 180,E1 -14802.97,E2 -14802.97} C_VEL
LIN {X 0,Y 326.571,Z 894.615,A -85,B 0,C 180,E1 -14807.029,E2 -14807.029} C_VEL
LIN {X 0,Y 326.57,Z 894.616,A -85,B 0,C 180,E1 -14810.781,E2 -14810.781} C_VEL
LIN {X 0,Y 326.61,Z 894.616,A -85,B 0,C 180,E1 -14814.48,E2 -14814.48} C_VEL
LIN {X 0,Y 326.607,Z 894.61,A -85,B 0,C 180,E1 -14817.455,E2 -14817.455} C_VEL
LIN {X 0,Y 326.614,Z 894.612,A -85,B 0,C 180,E1 -14820.336,E2 -14820.336} C_VEL
LIN {X 0,Y 326.656,Z 894.748,A -85,B 0,C 180,E1 -14822.49,E2 -14822.49} C_VEL
LIN {X 0,Y 328.759,Z 906.098,A -85,B 0,C 180,E1 -14826.035,E2 -14826.035} C_VEL
LIN {X 0,Y 328.774,Z 909.549,A -85,B 0,C 180,E1 -14827.067,E2 -14827.067} C_VEL
LIN {X 0,Y 327.409,Z 923.753,A -85,B 0,C 180,E1 -14831.217,E2 -14831.217} C_VEL
LIN {X 0,Y 327.087,Z 926.91,A -85,B 0,C 180,E1 -14832.13,E2 -14832.13} C_VEL
LIN {X 0,Y 329.769,Z 953.528,A -85,B 0,C 180,E1 -14833.055,E2 -14833.055} C_VEL
LIN {X 0,Y 330.244,Z 960.037,A -85,B 0,C 180,E1 -14833.266,E2 -14833.266} C_VEL
LIN {X 0,Y 329.249,Z 1005.781,A -85,B 0,C 180,E1 -14834.644,E2 -14834.644} C_VEL
LIN {X 0,Y 328.585,Z 1017.439,A -85,B 0,C 180,E1 -14835.207,E2 -14835.207} C_VEL
LIN {X 0,Y 328.234,Z 1027.245,A -85,B 0,C 180,E1 -14835.903,E2 -14835.903} C_VEL
LIN {X 0,Y 327.653,Z 1035.739,A -85,B 0,C 180,E1 -14836.668,E2 -14836.668} C_VEL
LIN {X 0,Y 327.125,Z 1044,A -85,B 0,C 180,E1 -14837.593,E2 -14837.593} C_VEL
LIN {X 0,Y 326.603,Z 1051.902,A -85,B 0,C 180,E1 -14838.676,E2 -14838.676} C_VEL
LIN {X 0,Y 325.974,Z 1060.196,A -85,B 0,C 180,E1 -14840.068,E2 -14840.068} C_VEL
LIN {X 0,Y 325.555,Z 1067.466,A -85,B 0,C 180,E1 -14841.621,E2 -14841.621} C_VEL
LIN {X 0,Y 325.323,Z 1073.197,A -85,B 0,C 180,E1 -14843.176,E2 -14843.176} C_VEL
LIN {X 0,Y 325.102,Z 1078.488,A -85,B 0,C 180,E1 -14845.039,E2 -14845.039} C_VEL
LIN {X 0,Y 324.943,Z 1082.277,A -85,B 0,C 180,E1 -14846.9,E2 -14846.9} C_VEL
LIN {X 0,Y 324.993,Z 1084.593,A -85,B 0,C 180,E1 -14848.761,E2 -14848.761} C_VEL
LIN {X 0,Y 325.019,Z 1085.496,A -85,B 0,C 180,E1 -14850,E2 -14850} C_VEL
LIN {X 0,Y 324.898,Z 1085.762,A -85,B 0,C 180,E1 -14851.239,E2 -14851.239} C_VEL
LIN {X 0,Y 324.877,Z 1085.458,A -85,B 0,C 180,E1 -14852.479,E2 -14852.479} C_VEL
LIN {X 0,Y 324.98,Z 1084.637,A -85,B 0,C 180,E1 -14853.72,E2 -14853.72} C_VEL
LIN {X 0,Y 325.013,Z 1083.292,A -85,B 0,C 180,E1 -14854.962,E2 -14854.962} C_VEL
LIN {X 0,Y 325.112,Z 1081.412,A -85,B 0,C 180,E1 -14856.205,E2 -14856.205} C_VEL
LIN {X 0,Y 325.567,Z 1077.343,A -85,B 0,C 180,E1 -14858.066,E2 -14858.066} C_VEL
LIN {X 0,Y 326.249,Z 1071.829,A -85,B 0,C 180,E1 -14859.923,E2 -14859.923} C_VEL
LIN {X 0,Y 327.043,Z 1065.941,A -85,B 0,C 180,E1 -14861.465,E2 -14861.465} C_VEL
LIN {X 0,Y 328.105,Z 1058.568,A -85,B 0,C 180,E1 -14862.997,E2 -14862.997} C_VEL
LIN {X 0,Y 329.218,Z 1050.294,A -85,B 0,C 180,E1 -14864.369,E2 -14864.369} C_VEL
LIN {X 0,Y 330.242,Z 1042.486,A -85,B 0,C 180,E1 -14865.427,E2 -14865.427} C_VEL
LIN {X 0,Y 331.213,Z 1034.411,A -85,B 0,C 180,E1 -14866.329,E2 -14866.329} C_VEL
LIN {X 0,Y 332.429,Z 1024.419,A -85,B 0,C 180,E1 -14867.216,E2 -14867.216} C_VEL
LIN {X 0,Y 333.63,Z 1012.671,A -85,B 0,C 180,E1 -14867.983,E2 -14867.983} C_VEL
LIN {X 0,Y 334.45,Z 1001.389,A -85,B 0,C 180,E1 -14868.499,E2 -14868.499} C_VEL
LIN {X 0,Y 336.379,Z 959.354,A -85,B 0,C 180,E1 -14869.918,E2 -14869.918} C_VEL
LIN {X 0,Y 335.285,Z 947.854,A -85,B 0,C 180,E1 -14870.486,E2 -14870.486} C_VEL
LIN {X 0,Y 332.89,Z 935.223,A -85,B 0,C 180,E1 -14871.282,E2 -14871.282} C_VEL
LIN {X 0,Y 329.993,Z 923.485,A -85,B 0,C 180,E1 -14872.152,E2 -14872.152} C_VEL
LIN {X 0,Y 330.975,Z 917.754,A -85,B 0,C 180,E1 -14874.068,E2 -14874.068} C_VEL
LIN {X 0,Y 330.765,Z 913.105,A -85,B 0,C 180,E1 -14875.822,E2 -14875.822} C_VEL
LIN {X 0,Y 329.348,Z 905.832,A -85,B 0,C 180,E1 -14878.967,E2 -14878.967} C_VEL
LIN {X 0,Y 328.188,Z 900.463,A -85,B 0,C 180,E1 -14881.644,E2 -14881.644} C_VEL
LIN {X 0,Y 326.633,Z 894.612,A -85,B 0,C 180,E1 -14885.19,E2 -14885.19} C_VEL
LIN {X 0,Y 326.564,Z 894.621,A -85,B 0,C 180,E1 -14888.617,E2 -14888.617} C_VEL
LIN {X 0,Y 326.558,Z 894.62,A -85,B 0,C 180,E1 -14891.848,E2 -14891.848} C_VEL
LIN {X 0,Y 326.522,Z 894.624,A -85,B 0,C 180,E1 -14895.258,E2 -14895.258} C_VEL
LIN {X 0,Y 326.558,Z 894.621,A -85,B 0,C 180,E1 -14898.152,E2 -14898.152} C_VEL
LIN {X 0,Y 326.564,Z 894.62,A -85,B 0,C 180,E1 -14901.384,E2 -14901.384} C_VEL
LIN {X 0,Y 326.615,Z 894.613,A -85,B 0,C 180,E1 -14904.852,E2 -14904.852} C_VEL
LIN {X 0,Y 326.606,Z 894.616,A -85,B 0,C 180,E1 -14907.456,E2 -14907.456} C_VEL
LIN {X 0,Y 326.598,Z 894.74,A -85,B 0,C 180,E1 -14911.042,E2 -14911.042} C_VEL
LIN {X 0,Y 327.949,Z 900.04,A -85,B 0,C 180,E1 -14914.622,E2 -14914.622} C_VEL
LIN {X 0,Y 329.102,Z 905.723,A -85,B 0,C 180,E1 -14917.817,E2 -14917.817} C_VEL
LIN {X 0,Y 330.99,Z 909.459,A -85,B 0,C 180,E1 -14918.241,E2 -14918.241} C_VEL
LIN {X 0,Y 335.366,Z 918.892,A -85,B 0,C 180,E1 -14919.188,E2 -14919.188} C_VEL
LIN {X 0,Y 337.601,Z 927.555,A -85,B 0,C 180,E1 -14919.81,E2 -14919.81} C_VEL
LIN {X 0,Y 334.691,Z 983.449,A -85,B 0,C 180,E1 -14921.72,E2 -14921.72} C_VEL
LIN {X 0,Y 333.887,Z 995.206,A -85,B 0,C 180,E1 -14922.388,E2 -14922.388} C_VEL
LIN {X 0,Y 332.978,Z 1004.908,A -85,B 0,C 180,E1 -14923.13,E2 -14923.13} C_VEL
LIN {X 0,Y 332.018,Z 1014.119,A -85,B 0,C 180,E1 -14924.028,E2 -14924.028} C_VEL
LIN {X 0,Y 330.714,Z 1024.857,A -85,B 0,C 180,E1 -14925.384,E2 -14925.384} C_VEL
LIN {X 0,Y 329.8,Z 1031.548,A -85,B 0,C 180,E1 -14926.444,E2 -14926.444} C_VEL
LIN {X 0,Y 328.889,Z 1037.909,A -85,B 0,C 180,E1 -14927.662,E2 -14927.662} C_VEL
LIN {X 0,Y 327.948,Z 1043.234,A -85,B 0,C 180,E1 -14928.88,E2 -14928.88} C_VEL
LIN {X 0,Y 327.311,Z 1047.672,A -85,B 0,C 180,E1 -14930.109,E2 -14930.109} C_VEL
LIN {X 0,Y 326.554,Z 1052.725,A -85,B 0,C 180,E1 -14931.89,E2 -14931.89} C_VEL
LIN {X 0,Y 326.035,Z 1055.546,A -85,B 0,C 180,E1 -14933.192,E2 -14933.192} C_VEL
LIN {X 0,Y 325.778,Z 1056.713,A -85,B 0,C 180,E1 -14933.808,E2 -14933.808} C_VEL
LIN {X 0,Y 325.436,Z 1058.418,A -85,B 0,C 180,E1 -14935.045,E2 -14935.045} C_VEL
LIN {X 0,Y 325.302,Z 1059.581,A -85,B 0,C 180,E1 -14936.284,E2 -14936.284} C_VEL
LIN {X 0,Y 325.175,Z 1060.236,A -85,B 0,C 180,E1 -14937.523,E2 -14937.523} C_VEL
LIN {X 0,Y 325.035,Z 1060.389,A -85,B 0,C 180,E1 -14938.762,E2 -14938.762} C_VEL
LIN {X 0,Y 324.95,Z 1059.953,A -85,B 0,C 180,E1 -14940.001,E2 -14940.001} C_VEL
LIN {X 0,Y 324.918,Z 1058.915,A -85,B 0,C 180,E1 -14941.24,E2 -14941.24} C_VEL
LIN {X 0,Y 325.007,Z 1056.425,A -85,B 0,C 180,E1 -14943.1,E2 -14943.1} C_VEL
LIN {X 0,Y 325.215,Z 1052.481,A -85,B 0,C 180,E1 -14944.96,E2 -14944.96} C_VEL
LIN {X 0,Y 325.407,Z 1047.957,A -85,B 0,C 180,E1 -14946.543,E2 -14946.543} C_VEL
LIN {X 0,Y 325.763,Z 1042.454,A -85,B 0,C 180,E1 -14948.062,E2 -14948.062} C_VEL
LIN {X 0,Y 326.189,Z 1035.439,A -85,B 0,C 180,E1 -14949.613,E2 -14949.613} C_VEL
LIN {X 0,Y 326.87,Z 1026.482,A -85,B 0,C 180,E1 -14951.158,E2 -14951.158} C_VEL
LIN {X 0,Y 327.373,Z 1018.685,A -85,B 0,C 180,E1 -14952.24,E2 -14952.24} C_VEL
LIN {X 0,Y 327.899,Z 1010.587,A -85,B 0,C 180,E1 -14953.164,E2 -14953.164} C_VEL
LIN {X 0,Y 328.299,Z 1002.301,A -85,B 0,C 180,E1 -14953.936,E2 -14953.936} C_VEL
LIN {X 0,Y 328.832,Z 991.796,A -85,B 0,C 180,E1 -14954.703,E2 -14954.703} C_VEL
LIN {X 0,Y 329.184,Z 979.664,A -85,B 0,C 180,E1 -14955.32,E2 -14955.32} C_VEL
LIN {X 0,Y 329.95,Z 950.448,A -85,B 0,C 180,E1 -14956.209,E2 -14956.209} C_VEL
LIN {X 0,Y 330.418,Z 922.596,A -85,B 0,C 180,E1 -14957.031,E2 -14957.031} C_VEL
LIN {X 0,Y 327.241,Z 901.102,A -85,B 0,C 180,E1 -14957.821,E2 -14957.821} C_VEL
LIN {X 0,Y 327.035,Z 896.547,A -85,B 0,C 180,E1 -14959.449,E2 -14959.449} C_VEL
LIN {X 0,Y 326.767,Z 894.592,A -85,B 0,C 180,E1 -14960.211,E2 -14960.211} C_VEL
LIN {X 0,Y 326.584,Z 894.613,A -85,B 0,C 180,E1 -14964.135,E2 -14964.135} C_VEL
LIN {X 0,Y 326.595,Z 894.611,A -85,B 0,C 180,E1 -14968.257,E2 -14968.257} C_VEL
LIN {X 0,Y 326.574,Z 894.617,A -85,B 0,C 180,E1 -14971.098,E2 -14971.098} C_VEL
LIN {X 0,Y 326.608,Z 894.611,A -85,B 0,C 180,E1 -14974.02,E2 -14974.02} C_VEL
LIN {X 0,Y 326.624,Z 894.61,A -85,B 0,C 180,E1 -14977.238,E2 -14977.238} C_VEL
LIN {X 0,Y 326.545,Z 894.618,A -85,B 0,C 180,E1 -14981.125,E2 -14981.125} C_VEL
LIN {X 0,Y 326.561,Z 894.618,A -85,B 0,C 180,E1 -14983.527,E2 -14983.527} C_VEL
LIN {X 0,Y 326.574,Z 894.614,A -85,B 0,C 180,E1 -14987.03,E2 -14987.03} C_VEL
LIN {X 0,Y 326.573,Z 894.616,A -85,B 0,C 180,E1 -14990.782,E2 -14990.782} C_VEL
LIN {X 0,Y 326.614,Z 894.615,A -85,B 0,C 180,E1 -14994.481,E2 -14994.481} C_VEL
LIN {X 0,Y 326.611,Z 894.609,A -85,B 0,C 180,E1 -14997.456,E2 -14997.456} C_VEL
LIN {X 0,Y 326.617,Z 894.612,A -85,B 0,C 180,E1 -15000.337,E2 -15000.337} C_VEL
LIN {X 0,Y 326.644,Z 894.609,A -85,B 0,C 180,E1 -15004.646,E2 -15004.646} C_VEL
LIN {X 0,Y 326.612,Z 894.611,A -85,B 0,C 180,E1 -15008.543,E2 -15008.543} C_VEL
LIN {X 0,Y 326.644,Z 894.606,A -85,B 0,C 180,E1 -15012.469,E2 -15012.469} C_VEL
LIN {X 0,Y 326.76,Z 894.591,A -85,B 0,C 180,E1 -15016.315,E2 -15016.315} C_VEL
LIN {X 0,Y 326.785,Z 894.589,A -85,B 0,C 180,E1 -15020.093,E2 -15020.093} C_VEL
LIN {X 0,Y 326.944,Z 894.573,A -85,B 0,C 180,E1 -15023.83,E2 -15023.83} C_VEL
LIN {X 0,Y 326.986,Z 894.566,A -85,B 0,C 180,E1 -15027.537,E2 -15027.537} C_VEL
LIN {X 0,Y 327.03,Z 894.557,A -85,B 0,C 180,E1 -15031.232,E2 -15031.232} C_VEL
LIN {X 0,Y 326.729,Z 894.597,A -85,B 0,C 180,E1 -15033.7,E2 -15033.7} C_VEL
LIN {X 0,Y 326.944,Z 894.573,A -85,B 0,C 180,E1 -15036.17,E2 -15036.17} C_VEL
LIN {X 0,Y 326.785,Z 894.589,A -85,B 0,C 180,E1 -15039.907,E2 -15039.907} C_VEL
LIN {X 0,Y 326.737,Z 894.594,A -85,B 0,C 180,E1 -15043.687,E2 -15043.687} C_VEL
LIN {X 0,Y 326.633,Z 894.607,A -85,B 0,C 180,E1 -15047.532,E2 -15047.532} C_VEL
LIN {X 0,Y 326.612,Z 894.611,A -85,B 0,C 180,E1 -15051.457,E2 -15051.457} C_VEL
LIN {X 0,Y 326.604,Z 894.613,A -85,B 0,C 180,E1 -15055.491,E2 -15055.491} C_VEL
LIN {X 0,Y 326.618,Z 894.612,A -85,B 0,C 180,E1 -15059.664,E2 -15059.664} C_VEL
LIN {X 0,Y 326.622,Z 894.61,A -85,B 0,C 180,E1 -15062.946,E2 -15062.946} C_VEL
LIN {X 0,Y 326.615,Z 894.615,A -85,B 0,C 180,E1 -15065.52,E2 -15065.52} C_VEL
LIN {X 0,Y 326.575,Z 894.615,A -85,B 0,C 180,E1 -15069.218,E2 -15069.218} C_VEL
LIN {X 0,Y 326.575,Z 894.614,A -85,B 0,C 180,E1 -15072.971,E2 -15072.971} C_VEL
LIN {X 0,Y 326.575,Z 894.614,A -85,B 0,C 180,E1 -15077.029,E2 -15077.029} C_VEL
LIN {X 0,Y 326.575,Z 894.615,A -85,B 0,C 180,E1 -15080.781,E2 -15080.781} C_VEL
LIN {X 0,Y 326.615,Z 894.615,A -85,B 0,C 180,E1 -15084.48,E2 -15084.48} C_VEL
LIN {X 0,Y 326.612,Z 894.609,A -85,B 0,C 180,E1 -15087.455,E2 -15087.455} C_VEL
LIN {X 0,Y 326.618,Z 894.612,A -85,B 0,C 180,E1 -15090.336,E2 -15090.336} C_VEL
LIN {X 0,Y 326.603,Z 894.613,A -85,B 0,C 180,E1 -15094.508,E2 -15094.508} C_VEL
LIN {X 0,Y 326.598,Z 894.615,A -85,B 0,C 180,E1 -15094.627,E2 -15094.627} C_VEL
LIN {X 0,Y 325.912,Z 894.707,A -85,B 0,C 180,E1 -15095.657,E2 -15095.657} C_VEL
LIN {X 0,Y 323.054,Z 895.063,A -85,B 0,C 180,E1 -15097.333,E2 -15097.333} C_VEL
LIN {X 0,Y 320.65,Z 895.356,A -85,B 0,C 180,E1 -15098.691,E2 -15098.691} C_VEL
LIN {X 0,Y 319.63,Z 895.48,A -85,B 0,C 180,E1 -15099.742,E2 -15099.742} C_VEL
LIN {X 0,Y 319.552,Z 895.489,A -85,B 0,C 180,E1 -15100.098,E2 -15100.098} C_VEL
LIN {X 0,Y 319.598,Z 895.488,A -85,B 0,C 180,E1 -15103.388,E2 -15103.388} C_VEL
LIN {X 0,Y 319.703,Z 895.471,A -85,B 0,C 180,E1 -15106.006,E2 -15106.006} C_VEL
LIN {X 0,Y 319.736,Z 895.469,A -85,B 0,C 180,E1 -15109.872,E2 -15109.872} C_VEL
LIN {X 0,Y 319.9,Z 895.452,A -85,B 0,C 180,E1 -15113.693,E2 -15113.693} C_VEL
LIN {X 0,Y 319.996,Z 895.434,A -85,B 0,C 180,E1 -15118.741,E2 -15118.741} C_VEL
LIN {X 0,Y 319.931,Z 895.444,A -85,B 0,C 180,E1 -15122.517,E2 -15122.517} C_VEL
LIN {X 0,Y 319.899,Z 895.452,A -85,B 0,C 180,E1 -15126.306,E2 -15126.306} C_VEL
LIN {X 0,Y 319.735,Z 895.469,A -85,B 0,C 180,E1 -15130.127,E2 -15130.127} C_VEL
LIN {X 0,Y 319.702,Z 895.471,A -85,B 0,C 180,E1 -15133.993,E2 -15133.993} C_VEL
LIN {X 0,Y 319.586,Z 895.485,A -85,B 0,C 180,E1 -15137.931,E2 -15137.931} C_VEL
LIN {X 0,Y 319.563,Z 895.487,A -85,B 0,C 180,E1 -15141.954,E2 -15141.954} C_VEL
LIN {X 0,Y 319.55,Z 895.489,A -85,B 0,C 180,E1 -15146.095,E2 -15146.095} C_VEL
LIN {X 0,Y 319.54,Z 895.493,A -85,B 0,C 180,E1 -15148.938,E2 -15148.938} C_VEL
LIN {X 0,Y 319.524,Z 895.494,A -85,B 0,C 180,E1 -15151.862,E2 -15151.862} C_VEL
LIN {X 0,Y 319.578,Z 895.492,A -85,B 0,C 180,E1 -15155.542,E2 -15155.542} C_VEL
LIN {X 0,Y 319.528,Z 895.497,A -85,B 0,C 180,E1 -15159.661,E2 -15159.661} C_VEL
LIN {X 0,Y 319.518,Z 895.495,A -85,B 0,C 180,E1 -15163.459,E2 -15163.459} C_VEL
LIN {X 0,Y 319.549,Z 895.489,A -85,B 0,C 180,E1 -15167.015,E2 -15167.015} C_VEL
LIN {X 0,Y 319.513,Z 895.499,A -85,B 0,C 180,E1 -15170.365,E2 -15170.365} C_VEL
LIN {X 0,Y 319.578,Z 895.492,A -85,B 0,C 180,E1 -15174.457,E2 -15174.457} C_VEL
LIN {X 0,Y 319.523,Z 895.495,A -85,B 0,C 180,E1 -15178.137,E2 -15178.137} C_VEL
LIN {X 0,Y 319.594,Z 895.484,A -85,B 0,C 180,E1 -15181.932,E2 -15181.932} C_VEL
LIN {X 0,Y 319.601,Z 895.591,A -85,B 0,C 180,E1 -15182.356,E2 -15182.356} C_VEL
LIN {X 0,Y 321.416,Z 905.238,A -85,B 0,C 180,E1 -15185.452,E2 -15185.452} C_VEL
LIN {X 0,Y 321.855,Z 908.623,A -85,B 0,C 180,E1 -15186.506,E2 -15186.506} C_VEL
LIN {X 0,Y 320.642,Z 920.583,A -85,B 0,C 180,E1 -15190.089,E2 -15190.089} C_VEL
LIN {X 0,Y 320.034,Z 926.899,A -85,B 0,C 180,E1 -15191.929,E2 -15191.929} C_VEL
LIN {X 0,Y 323.081,Z 956.647,A -85,B 0,C 180,E1 -15192.964,E2 -15192.964} C_VEL
LIN {X 0,Y 323.141,Z 964.88,A -85,B 0,C 180,E1 -15193.224,E2 -15193.224} C_VEL
LIN {X 0,Y 322.195,Z 1005.528,A -85,B 0,C 180,E1 -15194.502,E2 -15194.502} C_VEL
LIN {X 0,Y 321.503,Z 1017.66,A -85,B 0,C 180,E1 -15195.116,E2 -15195.116} C_VEL
LIN {X 0,Y 321.084,Z 1028.22,A -85,B 0,C 180,E1 -15195.906,E2 -15195.906} C_VEL
LIN {X 0,Y 320.547,Z 1036.469,A -85,B 0,C 180,E1 -15196.69,E2 -15196.69} C_VEL
LIN {X 0,Y 319.971,Z 1044.543,A -85,B 0,C 180,E1 -15197.634,E2 -15197.634} C_VEL
LIN {X 0,Y 319.367,Z 1053.353,A -85,B 0,C 180,E1 -15198.898,E2 -15198.898} C_VEL
LIN {X 0,Y 318.792,Z 1062.007,A -85,B 0,C 180,E1 -15200.483,E2 -15200.483} C_VEL
LIN {X 0,Y 318.453,Z 1067.604,A -85,B 0,C 180,E1 -15201.752,E2 -15201.752} C_VEL
LIN {X 0,Y 318.277,Z 1072.266,A -85,B 0,C 180,E1 -15203.024,E2 -15203.024} C_VEL
LIN {X 0,Y 318.029,Z 1076.415,A -85,B 0,C 180,E1 -15204.418,E2 -15204.418} C_VEL
LIN {X 0,Y 318.026,Z 1079.235,A -85,B 0,C 180,E1 -15205.564,E2 -15205.564} C_VEL
LIN {X 0,Y 317.837,Z 1082.571,A -85,B 0,C 180,E1 -15207.465,E2 -15207.465} C_VEL
LIN {X 0,Y 317.9,Z 1084.135,A -85,B 0,C 180,E1 -15208.733,E2 -15208.733} C_VEL
LIN {X 0,Y 317.929,Z 1085.084,A -85,B 0,C 180,E1 -15210,E2 -15210} C_VEL
LIN {X 0,Y 317.805,Z 1085.399,A -85,B 0,C 180,E1 -15211.267,E2 -15211.267} C_VEL
LIN {X 0,Y 317.799,Z 1085.196,A -85,B 0,C 180,E1 -15212.535,E2 -15212.535} C_VEL
LIN {X 0,Y 317.887,Z 1084.481,A -85,B 0,C 180,E1 -15213.803,E2 -15213.803} C_VEL
LIN {X 0,Y 317.926,Z 1083.244,A -85,B 0,C 180,E1 -15215.073,E2 -15215.073} C_VEL
LIN {X 0,Y 318.207,Z 1080.214,A -85,B 0,C 180,E1 -15216.977,E2 -15216.977} C_VEL
LIN {X 0,Y 318.717,Z 1075.848,A -85,B 0,C 180,E1 -15218.879,E2 -15218.879} C_VEL
LIN {X 0,Y 319.636,Z 1070.045,A -85,B 0,C 180,E1 -15220.771,E2 -15220.771} C_VEL
LIN {X 0,Y 320.574,Z 1063.756,A -85,B 0,C 180,E1 -15222.342,E2 -15222.342} C_VEL
LIN {X 0,Y 321.441,Z 1057.649,A -85,B 0,C 180,E1 -15223.594,E2 -15223.594} C_VEL
LIN {X 0,Y 322.699,Z 1049.235,A -85,B 0,C 180,E1 -15224.988,E2 -15224.988} C_VEL
LIN {X 0,Y 323.983,Z 1040.037,A -85,B 0,C 180,E1 -15226.218,E2 -15226.218} C_VEL
LIN {X 0,Y 325.28,Z 1030.081,A -85,B 0,C 180,E1 -15227.282,E2 -15227.282} C_VEL
LIN {X 0,Y 326.596,Z 1019.821,A -85,B 0,C 180,E1 -15228.1,E2 -15228.1} C_VEL
LIN {X 0,Y 327.668,Z 1009.475,A -85,B 0,C 180,E1 -15228.727,E2 -15228.727} C_VEL
LIN {X 0,Y 328.521,Z 997.487,A -85,B 0,C 180,E1 -15229.245,E2 -15229.245} C_VEL
LIN {X 0,Y 330.295,Z 960.186,A -85,B 0,C 180,E1 -15230.535,E2 -15230.535} C_VEL
LIN {X 0,Y 329.276,Z 948.85,A -85,B 0,C 180,E1 -15231.132,E2 -15231.132} C_VEL
LIN {X 0,Y 326.64,Z 935.369,A -85,B 0,C 180,E1 -15232.039,E2 -15232.039} C_VEL
LIN {X 0,Y 323.602,Z 922.995,A -85,B 0,C 180,E1 -15233.054,E2 -15233.054} C_VEL
LIN {X 0,Y 324.225,Z 919.023,A -85,B 0,C 180,E1 -15234.44,E2 -15234.44} C_VEL
LIN {X 0,Y 323.855,Z 914.16,A -85,B 0,C 180,E1 -15236.377,E2 -15236.377} C_VEL
LIN {X 0,Y 322.571,Z 907.612,A -85,B 0,C 180,E1 -15239.368,E2 -15239.368} C_VEL
LIN {X 0,Y 321.249,Z 901.884,A -85,B 0,C 180,E1 -15242.411,E2 -15242.411} C_VEL
LIN {X 0,Y 319.901,Z 896.963,A -85,B 0,C 180,E1 -15245.624,E2 -15245.624} C_VEL
LIN {X 0,Y 319.561,Z 895.492,A -85,B 0,C 180,E1 -15246.82,E2 -15246.82} C_VEL
LIN {X 0,Y 319.526,Z 895.497,A -85,B 0,C 180,E1 -15249.662,E2 -15249.662} C_VEL
LIN {X 0,Y 319.516,Z 895.497,A -85,B 0,C 180,E1 -15253.46,E2 -15253.46} C_VEL
LIN {X 0,Y 319.547,Z 895.492,A -85,B 0,C 180,E1 -15257.016,E2 -15257.016} C_VEL
LIN {X 0,Y 319.512,Z 895.496,A -85,B 0,C 180,E1 -15260.366,E2 -15260.366} C_VEL
LIN {X 0,Y 319.576,Z 895.492,A -85,B 0,C 180,E1 -15264.458,E2 -15264.458} C_VEL
LIN {X 0,Y 319.522,Z 895.497,A -85,B 0,C 180,E1 -15268.138,E2 -15268.138} C_VEL
LIN {X 0,Y 319.569,Z 895.541,A -85,B 0,C 180,E1 -15269.478,E2 -15269.478} C_VEL
LIN {X 0,Y 320.547,Z 899.565,A -85,B 0,C 180,E1 -15272.586,E2 -15272.586} C_VEL
LIN {X 0,Y 321.628,Z 903.941,A -85,B 0,C 180,E1 -15275.47,E2 -15275.47} C_VEL
LIN {X 0,Y 322.144,Z 906.458,A -85,B 0,C 180,E1 -15276.858,E2 -15276.858} C_VEL
LIN {X 0,Y 323.956,Z 909.94,A -85,B 0,C 180,E1 -15277.286,E2 -15277.286} C_VEL
LIN {X 0,Y 328.479,Z 918.955,A -85,B 0,C 180,E1 -15278.34,E2 -15278.34} C_VEL
LIN {X 0,Y 330.611,Z 924.473,A -85,B 0,C 180,E1 -15278.848,E2 -15278.848} C_VEL
LIN {X 0,Y 331.692,Z 929.959,A -85,B 0,C 180,E1 -15279.216,E2 -15279.216} C_VEL
LIN {X 0,Y 328.488,Z 984.158,A -85,B 0,C 180,E1 -15281.134,E2 -15281.134} C_VEL
LIN {X 0,Y 327.673,Z 995.563,A -85,B 0,C 180,E1 -15281.8,E2 -15281.8} C_VEL
LIN {X 0,Y 326.767,Z 1004.363,A -85,B 0,C 180,E1 -15282.476,E2 -15282.476} C_VEL
LIN {X 0,Y 325.913,Z 1012.221,A -85,B 0,C 180,E1 -15283.237,E2 -15283.237} C_VEL
LIN {X 0,Y 324.985,Z 1019.98,A -85,B 0,C 180,E1 -15284.156,E2 -15284.156} C_VEL
LIN {X 0,Y 323.716,Z 1028.526,A -85,B 0,C 180,E1 -15285.382,E2 -15285.382} C_VEL
LIN {X 0,Y 322.322,Z 1037.793,A -85,B 0,C 180,E1 -15287.086,E2 -15287.086} C_VEL
LIN {X 0,Y 321.3,Z 1043.212,A -85,B 0,C 180,E1 -15288.327,E2 -15288.327} C_VEL
LIN {X 0,Y 320.392,Z 1048.668,A -85,B 0,C 180,E1 -15289.894,E2 -15289.894} C_VEL
LIN {X 0,Y 319.811,Z 1052.205,A -85,B 0,C 180,E1 -15291.152,E2 -15291.152} C_VEL
LIN {X 0,Y 319.03,Z 1056.246,A -85,B 0,C 180,E1 -15293.041,E2 -15293.041} C_VEL
LIN {X 0,Y 318.763,Z 1057.376,A -85,B 0,C 180,E1 -15293.671,E2 -15293.671} C_VEL
LIN {X 0,Y 318.39,Z 1059.013,A -85,B 0,C 180,E1 -15294.935,E2 -15294.935} C_VEL
LIN {X 0,Y 318.228,Z 1060.067,A -85,B 0,C 180,E1 -15296.202,E2 -15296.202} C_VEL
LIN {X 0,Y 318.089,Z 1060.612,A -85,B 0,C 180,E1 -15297.468,E2 -15297.468} C_VEL
LIN {X 0,Y 317.941,Z 1060.65,A -85,B 0,C 180,E1 -15298.734,E2 -15298.734} C_VEL
LIN {X 0,Y 317.854,Z 1060.16,A -85,B 0,C 180,E1 -15300.001,E2 -15300.001} C_VEL
LIN {X 0,Y 317.827,Z 1059.058,A -85,B 0,C 180,E1 -15301.268,E2 -15301.268} C_VEL
LIN {X 0,Y 317.935,Z 1056.392,A -85,B 0,C 180,E1 -15303.169,E2 -15303.169} C_VEL
LIN {X 0,Y 318.08,Z 1053.87,A -85,B 0,C 180,E1 -15304.436,E2 -15304.436} C_VEL
LIN {X 0,Y 318.294,Z 1048.752,A -85,B 0,C 180,E1 -15306.339,E2 -15306.339} C_VEL
LIN {X 0,Y 318.658,Z 1043.21,A -85,B 0,C 180,E1 -15307.924,E2 -15307.924} C_VEL
LIN {X 0,Y 318.954,Z 1037.769,A -85,B 0,C 180,E1 -15309.193,E2 -15309.193} C_VEL
LIN {X 0,Y 319.407,Z 1031.224,A -85,B 0,C 180,E1 -15310.459,E2 -15310.459} C_VEL
LIN {X 0,Y 320.096,Z 1022.252,A -85,B 0,C 180,E1 -15311.879,E2 -15311.879} C_VEL
LIN {X 0,Y 320.679,Z 1011.9,A -85,B 0,C 180,E1 -15313.143,E2 -15313.143} C_VEL
LIN {X 0,Y 321.225,Z 1003.88,A -85,B 0,C 180,E1 -15313.927,E2 -15313.927} C_VEL
LIN {X 0,Y 321.688,Z 994.843,A -85,B 0,C 180,E1 -15314.633,E2 -15314.633} C_VEL
LIN {X 0,Y 321.921,Z 984.876,A -85,B 0,C 180,E1 -15315.229,E2 -15315.229} C_VEL
LIN {X 0,Y 322.407,Z 972.158,A -85,B 0,C 180,E1 -15315.732,E2 -15315.732} C_VEL
